C07284=1082.092,-4.857,441.669,174.077,19.888,153.353
C07285=1082.085,-5.106,441.682,174.075,19.886,153.353
C07286=1082.080,-5.356,441.696,174.074,19.884,153.352
C07287=1082.073,-5.606,441.710,174.073,19.882,153.352
C07288=1082.068,-5.855,441.724,174.072,19.880,153.352
C07289=1082.061,-6.105,441.737,174.069,19.877,153.352
C07290=1082.056,-6.354,441.751,174.068,19.875,153.352
C07291=1082.050,-6.603,441.764,174.067,19.873,153.352
C07292=1082.044,-6.853,441.778,174.066,19.871,153.351
C07293=1082.037,-7.103,441.792,174.064,19.870,153.351
C07294=1082.032,-7.352,441.806,174.062,19.867,153.351
C07295=1082.026,-7.602,441.819,174.061,19.865,153.351
C07296=1082.020,-7.851,441.833,174.060,19.863,153.351
C07297=1082.015,-8.102,441.846,174.058,19.861,153.351
C07298=1082.009,-8.351,441.859,174.056,19.859,153.351
C07299=1082.003,-8.600,441.873,174.055,19.857,153.350
C07300=1081.997,-8.850,441.886,174.054,19.855,153.350
C07301=1081.991,-9.100,441.901,174.052,19.853,153.350
C07302=1081.985,-9.349,441.914,174.051,19.851,153.350
C07303=1081.979,-9.599,441.928,174.049,19.848,153.350
C07304=1081.973,-9.848,441.941,174.048,19.846,153.350
C07305=1081.968,-10.098,441.954,174.046,19.845,153.350
C07306=1081.962,-10.347,441.967,174.045,19.843,153.349
C07307=1081.956,-10.597,441.981,174.043,19.840,153.349
C07308=1081.950,-10.846,441.994,174.042,19.838,153.349
C07309=1081.945,-11.096,442.008,174.041,19.836,153.349
C07310=1081.938,-11.345,442.022,174.039,19.834,153.349
C07311=1081.932,-11.595,442.034,174.038,19.832,153.349
C07312=1081.927,-11.845,442.048,174.036,19.830,153.348
C07313=1081.920,-12.095,442.062,174.035,19.828,153.348
C07314=1081.915,-12.344,442.076,174.033,19.826,153.348
C07315=1081.908,-12.593,442.089,174.032,19.824,153.348
C07316=1081.903,-12.844,442.102,174.031,19.822,153.348
C07317=1081.897,-13.093,442.115,174.029,19.820,153.348
C07318=1081.892,-13.342,442.129,174.027,19.818,153.348
C07319=1081.885,-13.592,442.142,174.026,19.816,153.347
C07320=1081.880,-13.842,442.156,174.025,19.814,153.347
C07321=1081.874,-14.091,442.169,174.023,19.811,153.347
C07322=1081.869,-14.341,442.183,174.021,19.809,153.347
C07323=1081.862,-14.590,442.196,174.020,19.807,153.347
C07324=1081.856,-14.840,442.208,174.019,19.805,153.347
C07325=1081.851,-15.089,442.222,174.018,19.803,153.346
C07326=1081.845,-15.339,442.236,174.016,19.801,153.346
C07327=1081.839,-15.589,442.248,174.014,19.799,153.346
C07328=1081.833,-15.838,442.262,174.013,19.797,153.346
C07329=1081.827,-16.087,442.275,174.012,19.795,153.346
C07330=1081.821,-16.337,442.288,174.010,19.793,153.346
C07331=1081.816,-16.587,442.302,174.008,19.791,153.346
C07332=1081.809,-16.860,442.316,174.007,19.789,153.345
C07333=1081.802,-17.135,442.331,174.006,19.787,153.345
C07334=1081.796,-17.409,442.345,174.004,19.784,153.345
C07335=1081.789,-17.683,442.360,174.002,19.782,153.345
C07336=1081.783,-17.933,442.372,174.001,19.780,153.345
C07337=1081.777,-18.182,442.386,173.999,19.778,153.345
C07338=1081.772,-18.431,442.399,173.998,19.776,153.345
C07339=1081.766,-18.681,442.412,173.996,19.774,153.344
C07340=1081.760,-18.931,442.425,173.995,19.772,153.344
C07341=1081.754,-19.180,442.438,173.994,19.770,153.344
C07342=1081.748,-19.430,442.452,173.992,19.768,153.344
C07343=1081.742,-19.680,442.464,173.990,19.766,153.344
C07344=1081.736,-19.929,442.477,173.989,19.764,153.344
C07345=1081.730,-20.178,442.491,173.988,19.762,153.344
C07346=1081.724,-20.428,442.503,173.987,19.760,153.343
C07347=1081.719,-20.678,442.517,173.984,19.758,153.343
C07348=1081.713,-20.928,442.530,173.983,19.756,153.343
C07349=1081.706,-21.177,442.543,173.982,19.754,153.343
C07350=1081.701,-21.427,442.556,173.980,19.752,153.343
C07351=1081.695,-21.677,442.569,173.979,19.750,153.343
C07352=1081.689,-21.926,442.582,173.978,19.748,153.343
C07353=1081.683,-22.176,442.595,173.976,19.746,153.342
C07354=1081.677,-22.426,442.608,173.974,19.744,153.342
C07355=1081.671,-22.675,442.621,173.973,19.742,153.342
C07356=1081.666,-22.925,442.634,173.972,19.740,153.342
C07357=1081.659,-23.174,442.647,173.971,19.738,153.342
C07358=1081.654,-23.424,442.660,173.969,19.736,153.342
C07359=1081.647,-23.673,442.673,173.967,19.734,153.342
C07360=1081.642,-23.923,442.685,173.966,19.732,153.342
C07361=1081.636,-24.172,442.699,173.965,19.730,153.341
C07362=1081.631,-24.422,442.712,173.963,19.728,153.341
C07363=1081.625,-24.672,442.724,173.961,19.725,153.341
C07364=1081.618,-24.921,442.738,173.960,19.723,153.341
C07365=1081.613,-25.171,442.750,173.958,19.722,153.341
C07366=1081.606,-25.420,442.764,173.957,19.720,153.341
C07367=1081.600,-25.670,442.776,173.956,19.718,153.341
C07368=1081.595,-25.920,442.789,173.955,19.716,153.340
C07369=1081.590,-26.169,442.802,173.953,19.713,153.340
C07370=1081.584,-26.419,442.815,173.951,19.712,153.340
C07371=1081.578,-26.668,442.828,173.950,19.710,153.340
C07372=1081.572,-26.918,442.841,173.949,19.708,153.340
C07373=1081.566,-27.168,442.853,173.947,19.706,153.340
C07374=1081.560,-27.417,442.866,173.946,19.704,153.340
C07375=1081.554,-27.667,442.879,173.944,19.702,153.340
C07376=1081.548,-27.917,442.891,173.943,19.700,153.339
C07377=1081.541,-28.166,442.905,173.941,19.698,153.339
C07378=1081.536,-28.415,442.917,173.940,19.696,153.339
C07379=1081.530,-28.665,442.929,173.939,19.694,153.339
C07380=1081.524,-28.915,442.943,173.937,19.692,153.339
C07381=1081.518,-29.164,442.955,173.935,19.690,153.339
C07382=1081.512,-29.414,442.968,173.934,19.688,153.339
C07383=1081.506,-29.664,442.980,173.933,19.686,153.338
C07384=1081.500,-29.913,442.994,173.931,19.684,153.338
C07385=1081.494,-30.163,443.006,173.930,19.683,153.338
C07386=1081.488,-30.413,443.019,173.929,19.681,153.338
C07387=1081.483,-30.662,443.032,173.927,19.678,153.338
C07388=1081.477,-30.912,443.044,173.925,19.677,153.338
C07389=1081.471,-31.162,443.057,173.924,19.675,153.338
C07390=1081.465,-31.411,443.069,173.923,19.673,153.338
C07391=1081.459,-31.661,443.082,173.921,19.671,153.338
C07392=1081.452,-31.910,443.095,173.920,19.669,153.337
C07393=1081.447,-32.159,443.107,173.918,19.667,153.337
C07394=1081.441,-32.409,443.119,173.916,19.665,153.337
C07395=1081.435,-32.659,443.132,173.915,19.663,153.337
C07396=1081.428,-32.933,443.146,173.914,19.661,153.337
C07397=1081.422,-33.206,443.160,173.912,19.659,153.337
C07398=1081.416,-33.479,443.173,173.910,19.657,153.337
C07399=1081.409,-33.752,443.188,173.909,19.655,153.336
C07400=1081.403,-34.002,443.200,173.908,19.653,153.336
C07401=1081.398,-34.251,443.212,173.906,19.651,153.336
C07402=1081.392,-34.501,443.225,173.904,19.649,153.336
C07403=1081.386,-34.751,443.237,173.903,19.647,153.336
C07404=1081.379,-35.001,443.249,173.902,19.645,153.336
C07405=1081.373,-35.250,443.263,173.900,19.643,153.336
C07406=1081.368,-35.499,443.275,173.899,19.642,153.336
C07407=1081.362,-35.749,443.287,173.897,19.639,153.336
C07408=1081.356,-35.999,443.300,173.896,19.637,153.335
C07409=1081.350,-36.249,443.312,173.894,19.636,153.335
C07410=1081.345,-36.498,443.325,173.893,19.634,153.335
C07411=1081.339,-36.748,443.337,173.892,19.632,153.335
C07412=1081.333,-36.998,443.350,173.890,19.630,153.335
C07413=1081.326,-37.247,443.362,173.889,19.628,153.335
C07414=1081.321,-37.496,443.374,173.887,19.626,153.335
C07415=1081.315,-37.746,443.386,173.885,19.624,153.335
C07416=1081.309,-37.996,443.399,173.884,19.622,153.334
C07417=1081.303,-38.245,443.412,173.883,19.620,153.334
C07418=1081.298,-38.495,443.424,173.881,19.618,153.334
C07419=1081.291,-38.744,443.436,173.880,19.616,153.334
C07420=1081.285,-38.994,443.449,173.879,19.614,153.334
C07421=1081.279,-39.244,443.462,173.877,19.612,153.334
C07422=1081.274,-39.493,443.474,173.875,19.610,153.334
C07423=1081.267,-39.743,443.486,173.874,19.609,153.334
C07424=1081.261,-39.993,443.498,173.873,19.607,153.334
C07425=1081.255,-40.243,443.511,173.871,19.605,153.334
C07426=1081.249,-40.491,443.522,173.870,19.603,153.333
C07427=1081.243,-40.741,443.535,173.869,19.601,153.333
C07428=1081.238,-40.992,443.547,173.867,19.600,153.333
C07429=1081.231,-41.241,443.559,173.865,19.597,153.333
C07430=1081.226,-41.491,443.571,173.864,19.596,153.333
C07431=1081.220,-41.740,443.583,173.862,19.594,153.333
C07432=1081.213,-41.990,443.595,173.861,19.592,153.333
C07433=1081.207,-42.240,443.608,173.860,19.590,153.333
C07434=1081.202,-42.489,443.620,173.858,19.589,153.333
C07435=1081.195,-42.739,443.632,173.857,19.587,153.332
C07436=1081.190,-42.989,443.645,173.855,19.584,153.332
C07437=1081.184,-43.238,443.657,173.853,19.583,153.332
C07438=1081.178,-43.487,443.669,173.852,19.581,153.332
C07439=1081.172,-43.737,443.681,173.851,19.579,153.332
C07440=1081.167,-43.987,443.693,173.849,19.577,153.332
C07441=1081.160,-44.237,443.705,173.848,19.576,153.332
C07442=1081.154,-44.486,443.717,173.847,19.574,153.332
C07443=1081.148,-44.736,443.730,173.845,19.572,153.332
C07444=1081.142,-44.985,443.742,173.844,19.570,153.331
C07445=1081.136,-45.235,443.754,173.842,19.568,153.331
C07446=1081.130,-45.485,443.766,173.840,19.566,153.331
C07447=1081.125,-45.734,443.778,173.839,19.565,153.331
C07448=1081.119,-45.984,443.790,173.838,19.563,153.331
C07449=1081.112,-46.234,443.802,173.836,19.561,153.331
C07450=1081.107,-46.483,443.814,173.835,19.559,153.331
C07451=1081.100,-46.733,443.826,173.834,19.558,153.331
C07452=1081.095,-46.982,443.838,173.832,19.556,153.331
C07453=1081.089,-47.232,443.850,173.830,19.553,153.331
C07454=1081.083,-47.482,443.862,173.829,19.552,153.331
C07455=1081.077,-47.731,443.874,173.828,19.550,153.330
C07456=1081.072,-47.982,443.886,173.826,19.548,153.330
C07457=1081.065,-48.231,443.898,173.825,19.546,153.330
C07458=1081.060,-48.480,443.910,173.823,19.545,153.330
C07459=1081.053,-48.730,443.922,173.822,19.543,153.330
C07460=1081.047,-49.004,443.935,173.820,19.541,153.330
C07461=1081.040,-49.278,443.948,173.819,19.539,153.330
C07462=1081.034,-49.551,443.962,173.817,19.537,153.330
C07463=1081.027,-49.825,443.975,173.816,19.535,153.330
C07464=1081.022,-50.074,443.987,173.814,19.533,153.329
C07465=1081.016,-50.324,443.999,173.812,19.531,153.329
C07466=1081.011,-50.574,444.010,173.811,19.530,153.329
C07467=1081.004,-50.823,444.022,173.810,19.527,153.329
C07468=1080.997,-51.073,444.034,173.808,19.526,153.329
C07469=1080.992,-51.322,444.046,173.807,19.524,153.329
C07470=1080.986,-51.572,444.058,173.805,19.522,153.329
C07471=1080.979,-51.822,444.069,173.804,19.521,153.329
C07472=1080.974,-52.072,444.081,173.803,19.519,153.329
C07473=1080.967,-52.321,444.093,173.801,19.517,153.329
C07474=1080.961,-52.571,444.105,173.799,19.515,153.329
C07475=1080.955,-52.820,444.116,173.798,19.513,153.329
C07476=1080.949,-53.070,444.128,173.796,19.512,153.329
C07477=1080.942,-53.320,444.140,173.795,19.510,153.329
C07478=1080.937,-53.569,444.151,173.794,19.508,153.328
C07479=1080.931,-53.819,444.164,173.792,19.507,153.328
C07480=1080.925,-54.069,444.175,173.791,19.505,153.328
C07481=1080.918,-54.318,444.187,173.789,19.503,153.328
C07482=1080.912,-54.568,444.199,173.788,19.502,153.328
C07483=1080.907,-54.817,444.210,173.786,19.500,153.328
C07484=1080.900,-55.067,444.222,173.785,19.499,153.328
C07485=1080.894,-55.317,444.233,173.784,19.497,153.328
C07486=1080.888,-55.566,444.245,173.781,19.495,153.328
C07487=1080.882,-55.817,444.257,173.780,19.493,153.328
C07488=1080.876,-56.065,444.268,173.779,19.491,153.328
C07489=1080.870,-56.315,444.281,173.777,19.490,153.328
C07490=1080.864,-56.565,444.292,173.776,19.488,153.328
C07491=1080.858,-56.814,444.304,173.774,19.486,153.327
C07492=1080.851,-57.065,444.315,173.773,19.485,153.327
C07493=1080.846,-57.314,444.327,173.772,19.483,153.327
C07494=1080.840,-57.564,444.338,173.770,19.482,153.327
C07495=1080.834,-57.813,444.350,173.769,19.480,153.327
C07496=1080.827,-58.063,444.361,173.767,19.478,153.327
C07497=1080.822,-58.312,444.373,173.766,19.477,153.327
C07498=1080.816,-58.562,444.385,173.765,19.475,153.327
C07499=1080.810,-58.812,444.395,173.762,19.473,153.327
C07500=1080.803,-59.061,444.407,173.761,19.471,153.327
C07501=1080.798,-59.312,444.419,173.759,19.470,153.327
C07502=1080.792,-59.561,444.431,173.758,19.468,153.327
C07503=1080.785,-59.811,444.442,173.757,19.466,153.327
C07504=1080.779,-60.060,444.454,173.755,19.465,153.327
C07505=1080.774,-60.310,444.465,173.754,19.463,153.327
C07506=1080.768,-60.559,444.477,173.753,19.461,153.327
C07507=1080.761,-60.809,444.488,173.751,19.460,153.326
C07508=1080.756,-61.059,444.499,173.750,19.458,153.326
C07509=1080.750,-61.309,444.512,173.748,19.457,153.326
C07510=1080.744,-61.558,444.523,173.747,19.455,153.326
C07511=1080.737,-61.808,444.535,173.745,19.453,153.326
C07512=1080.731,-62.057,444.545,173.744,19.452,153.326
C07513=1080.725,-62.308,444.557,173.742,19.450,153.326
C07514=1080.720,-62.557,444.569,173.740,19.448,153.326
C07515=1080.713,-62.807,444.580,173.739,19.446,153.326
C07516=1080.708,-63.056,444.591,173.737,19.445,153.326
C07517=1080.702,-63.305,444.603,173.736,19.443,153.326
C07518=1080.695,-63.556,444.614,173.735,19.441,153.326
C07519=1080.690,-63.805,444.625,173.733,19.440,153.326
C07520=1080.684,-64.055,444.637,173.732,19.438,153.326
C07521=1080.678,-64.304,444.648,173.730,19.437,153.326
C07522=1080.672,-64.555,444.659,173.729,19.435,153.326
C07523=1080.666,-64.803,444.671,173.728,19.433,153.326
C07524=1080.660,-65.079,444.683,173.726,19.432,153.325
C07525=1080.653,-65.354,444.696,173.724,19.430,153.326
C07526=1080.646,-65.629,444.708,173.723,19.428,153.325
C07527=1080.640,-65.904,444.721,173.721,19.426,153.325
C07528=1080.634,-66.153,444.732,173.720,19.425,153.325
C07529=1080.627,-66.403,444.744,173.718,19.423,153.325
C07530=1080.622,-66.652,444.754,173.717,19.421,153.325
C07531=1080.615,-66.903,444.766,173.716,19.420,153.325
C07532=1080.610,-67.152,444.777,173.714,19.418,153.325
C07533=1080.604,-67.401,444.789,173.713,19.417,153.325
C07534=1080.598,-67.652,444.800,173.711,19.415,153.325
C07535=1080.592,-67.901,444.811,173.710,19.414,153.325
C07536=1080.586,-68.151,444.822,173.708,19.412,153.325
C07537=1080.580,-68.401,444.833,173.707,19.410,153.325
C07538=1080.574,-68.650,444.845,173.705,19.408,153.325
C07539=1080.568,-68.900,444.856,173.703,19.407,153.325
C07540=1080.563,-69.150,444.867,173.702,19.405,153.325
C07541=1080.557,-69.399,444.878,173.700,19.404,153.325
C07542=1080.551,-69.649,444.889,173.699,19.401,153.324
C07543=1080.545,-69.899,444.900,173.698,19.400,153.324
C07544=1080.539,-70.148,444.912,173.696,19.398,153.324
C07545=1080.533,-70.398,444.923,173.695,19.397,153.324
C07546=1080.527,-70.647,444.934,173.693,19.395,153.324
C07547=1080.521,-70.897,444.945,173.692,19.394,153.324
C07548=1080.515,-71.147,444.957,173.690,19.392,153.324
C07549=1080.510,-71.397,444.968,173.689,19.390,153.324
C07550=1080.504,-71.646,444.978,173.687,19.389,153.324
C07551=1080.498,-71.896,444.990,173.686,19.387,153.324
C07552=1080.492,-72.145,445.001,173.685,19.386,153.324
C07553=1080.486,-72.395,445.012,173.683,19.384,153.324
C07554=1080.479,-72.645,445.023,173.682,19.383,153.324
C07555=1080.474,-72.894,445.034,173.680,19.381,153.324
C07556=1080.468,-73.144,445.045,173.679,19.380,153.324
C07557=1080.462,-73.393,445.056,173.677,19.378,153.324
C07558=1080.456,-73.644,445.067,173.676,19.376,153.324
C07559=1080.451,-73.893,445.079,173.675,19.375,153.324
C07560=1080.445,-74.143,445.090,173.673,19.373,153.324
C07561=1080.438,-74.393,445.100,173.672,19.372,153.324
C07562=1080.432,-74.642,445.111,173.670,19.370,153.324
C07563=1080.427,-74.892,445.122,173.669,19.369,153.324
C07564=1080.420,-75.142,445.133,173.667,19.367,153.324
C07565=1080.415,-75.392,445.144,173.666,19.366,153.324
C07566=1080.409,-75.641,445.155,173.664,19.364,153.324
C07567=1080.402,-75.891,445.166,173.663,19.363,153.323
C07568=1080.397,-76.141,445.177,173.661,19.361,153.323
C07569=1080.390,-76.390,445.187,173.660,19.360,153.323
C07570=1080.384,-76.640,445.199,173.658,19.359,153.324
C07571=1080.378,-76.890,445.210,173.657,19.357,153.324
C07572=1080.372,-77.139,445.220,173.655,19.356,153.323
C07573=1080.366,-77.389,445.232,173.654,19.354,153.323
C07574=1080.360,-77.639,445.243,173.652,19.353,153.323
C07575=1080.355,-77.888,445.253,173.651,19.351,153.323
C07576=1080.349,-78.138,445.264,173.649,19.350,153.323
C07577=1080.342,-78.388,445.275,173.648,19.348,153.323
C07578=1080.336,-78.637,445.286,173.646,19.347,153.323
C07579=1080.330,-78.887,445.297,173.645,19.345,153.323
C07580=1080.324,-79.137,445.307,173.643,19.344,153.323
C07581=1080.319,-79.387,445.318,173.642,19.342,153.323
C07582=1080.313,-79.636,445.329,173.641,19.341,153.323
C07583=1080.306,-79.886,445.339,173.639,19.339,153.323
C07584=1080.300,-80.136,445.351,173.638,19.338,153.323
C07585=1080.294,-80.385,445.361,173.636,19.337,153.323
C07586=1080.289,-80.635,445.372,173.634,19.335,153.323
C07587=1080.281,-80.885,445.383,173.633,19.334,153.323
C07588=1080.276,-81.162,445.394,173.631,19.332,153.323
C07589=1080.268,-81.439,445.406,173.629,19.330,153.323
C07590=1080.261,-81.716,445.419,173.628,19.329,153.323
C07591=1080.255,-81.993,445.430,173.626,19.327,153.323
C07592=1080.248,-82.243,445.441,173.625,19.326,153.323
C07593=1080.243,-82.493,445.452,173.623,19.325,153.323
C07594=1080.236,-82.742,445.462,173.622,19.323,153.323
C07595=1080.230,-82.991,445.473,173.620,19.322,153.323
C07596=1080.224,-83.242,445.483,173.618,19.321,153.323
C07597=1080.218,-83.491,445.494,173.617,19.319,153.323
C07598=1080.212,-83.741,445.505,173.615,19.318,153.323
C07599=1080.206,-83.991,445.516,173.614,19.316,153.323
C07600=1080.199,-84.240,445.526,173.613,19.315,153.323
C07601=1080.194,-84.490,445.536,173.611,19.314,153.323
C07602=1080.188,-84.740,445.547,173.609,19.312,153.323
C07603=1080.181,-84.990,445.558,173.608,19.311,153.323
C07604=1080.175,-85.239,445.569,173.606,19.309,153.323
C07605=1080.169,-85.489,445.578,173.605,19.308,153.323
C07606=1080.164,-85.738,445.589,173.603,19.307,153.323
C07607=1080.157,-85.989,445.600,173.603,19.306,153.323
C07608=1080.151,-86.238,445.611,173.601,19.304,153.323
C07609=1080.145,-86.488,445.621,173.600,19.303,153.323
C07610=1080.139,-86.737,445.631,173.598,19.302,153.323
C07611=1080.133,-86.987,445.642,173.597,19.300,153.323
C07612=1080.127,-87.237,445.652,173.595,19.299,153.323
C07613=1080.121,-87.487,445.663,173.593,19.298,153.323
C07614=1080.115,-87.736,445.674,173.592,19.296,153.323
C07615=1080.109,-87.986,445.683,173.590,19.295,153.323
C07616=1080.103,-88.235,445.694,173.589,19.294,153.323
C07617=1080.097,-88.486,445.705,173.587,19.292,153.323
C07618=1080.090,-88.735,445.715,173.586,19.291,153.323
C07619=1080.085,-88.985,445.726,173.584,19.290,153.323
C07620=1080.078,-89.234,445.736,173.583,19.288,153.323
C07621=1080.073,-89.484,445.746,173.581,19.287,153.323
C07622=1080.066,-89.733,445.756,173.579,19.286,153.324
C07623=1080.060,-89.984,445.768,173.578,19.284,153.324
C07624=1080.054,-90.234,445.778,173.577,19.283,153.323
C07625=1080.048,-90.483,445.788,173.575,19.282,153.324
C07626=1080.043,-90.733,445.798,173.573,19.280,153.324
C07627=1080.036,-90.982,445.809,173.572,19.279,153.324
C07628=1080.030,-91.232,445.819,173.571,19.278,153.324
C07629=1080.024,-91.482,445.829,173.570,19.277,153.324
C07630=1080.018,-91.732,445.840,173.568,19.275,153.324
C07631=1080.012,-91.981,445.850,173.566,19.275,153.324
C07632=1080.006,-92.231,445.861,173.565,19.273,153.324
C07633=1080.000,-92.480,445.872,173.564,19.272,153.324
C07634=1079.994,-92.730,445.881,173.562,19.271,153.324
C07635=1079.988,-92.980,445.892,173.560,19.269,153.324
C07636=1079.982,-93.229,445.902,173.559,19.268,153.324
C07637=1079.976,-93.480,445.913,173.557,19.267,153.324
C07638=1079.970,-93.729,445.922,173.556,19.265,153.324
C07639=1079.964,-93.979,445.933,173.554,19.264,153.324
C07640=1079.958,-94.229,445.943,173.553,19.263,153.324
C07641=1079.952,-94.478,445.954,173.551,19.261,153.324
C07642=1079.946,-94.728,445.963,173.549,19.260,153.324
C07643=1079.940,-94.977,445.974,173.548,19.259,153.324
C07644=1079.934,-95.227,445.984,173.547,19.258,153.324
C07645=1079.928,-95.477,445.995,173.546,19.257,153.324
C07646=1079.922,-95.727,446.004,173.544,19.255,153.324
C07647=1079.916,-95.976,446.015,173.542,19.254,153.324
C07648=1079.910,-96.226,446.025,173.541,19.253,153.324
C07649=1079.905,-96.476,446.035,173.539,19.252,153.324
C07650=1079.898,-96.726,446.045,173.538,19.250,153.324
C07651=1079.892,-96.976,446.056,173.536,19.249,153.324
C07652=1079.885,-97.255,446.067,173.535,19.248,153.324
C07653=1079.879,-97.535,446.078,173.533,19.246,153.324
C07654=1079.872,-97.815,446.090,173.531,19.245,153.324
C07655=1079.865,-98.094,446.101,173.530,19.244,153.324
C07656=1079.859,-98.345,446.111,173.528,19.243,153.324
C07657=1079.853,-98.594,446.121,173.527,19.241,153.324
C07658=1079.847,-98.844,446.131,173.525,19.240,153.324
C07659=1079.840,-99.093,446.141,173.523,19.239,153.325
C07660=1079.835,-99.343,446.151,173.522,19.238,153.325
C07661=1079.828,-99.592,446.162,173.520,19.237,153.325
C07662=1079.822,-99.842,446.171,173.519,19.235,153.325
C07663=1079.816,-100.091,446.182,173.517,19.234,153.325
C07664=1079.810,-100.341,446.192,173.516,19.233,153.325
C07665=1079.804,-100.590,446.202,173.515,19.232,153.325
C07666=1079.798,-100.840,446.212,173.513,19.231,153.325
C07667=1079.791,-101.090,446.221,173.512,19.230,153.325
C07668=1079.786,-101.339,446.232,173.510,19.229,153.325
C07669=1079.780,-101.589,446.242,173.508,19.227,153.325
C07670=1079.773,-101.839,446.251,173.507,19.226,153.325
C07671=1079.768,-102.088,446.262,173.505,19.225,153.325
C07672=1079.761,-102.338,446.272,173.504,19.224,153.325
C07673=1079.755,-102.588,446.281,173.502,19.223,153.325
C07674=1079.749,-102.837,446.291,173.500,19.221,153.325
C07675=1079.743,-103.087,446.302,173.500,19.221,153.325
C07676=1079.737,-103.337,446.311,173.498,19.220,153.325
C07677=1079.731,-103.587,446.321,173.496,19.218,153.325
C07678=1079.725,-103.836,446.331,173.495,19.217,153.326
C07679=1079.719,-104.086,446.341,173.493,19.216,153.326
C07680=1079.713,-104.336,446.351,173.491,19.215,153.326
C07681=1079.707,-104.586,446.360,173.490,19.214,153.326
C07682=1079.700,-104.835,446.371,173.488,19.213,153.326
C07683=1079.695,-105.085,446.381,173.487,19.212,153.326
C07684=1079.689,-105.335,446.390,173.486,19.211,153.326
C07685=1079.683,-105.585,446.400,173.484,19.210,153.326
C07686=1079.676,-105.834,446.409,173.483,19.209,153.326
C07687=1079.671,-106.084,446.420,173.481,19.208,153.326
C07688=1079.664,-106.334,446.430,173.479,19.207,153.326
C07689=1079.658,-106.584,446.439,173.477,19.206,153.326
C07690=1079.652,-106.833,446.449,173.476,19.204,153.326
C07691=1079.646,-107.083,446.459,173.475,19.204,153.326
C07692=1079.640,-107.333,446.469,173.473,19.203,153.327
C07693=1079.634,-107.582,446.479,173.472,19.201,153.326
C07694=1079.628,-107.832,446.489,173.470,19.200,153.327
C07695=1079.622,-108.082,446.498,173.469,19.199,153.327
C07696=1079.616,-108.332,446.508,173.467,19.198,153.327
C07697=1079.609,-108.582,446.517,173.465,19.197,153.327
C07698=1079.603,-108.831,446.528,173.464,19.196,153.327
C07699=1079.597,-109.081,446.537,173.463,19.195,153.327
C07700=1079.591,-109.330,446.547,173.461,19.194,153.327
C07701=1079.585,-109.581,446.557,173.459,19.193,153.327
C07702=1079.579,-109.830,446.566,173.458,19.192,153.327
C07703=1079.573,-110.080,446.576,173.456,19.191,153.327
C07704=1079.567,-110.330,446.586,173.455,19.190,153.327
C07705=1079.560,-110.580,446.595,173.453,19.189,153.328
C07706=1079.554,-110.829,446.605,173.452,19.188,153.328
C07707=1079.548,-111.079,446.615,173.450,19.187,153.328
C07708=1079.542,-111.328,446.625,173.449,19.186,153.328
C07709=1079.535,-111.578,446.634,173.447,19.185,153.328
C07710=1079.529,-111.828,446.644,173.445,19.184,153.328
C07711=1079.524,-112.077,446.653,173.444,19.183,153.328
C07712=1079.518,-112.327,446.662,173.443,19.183,153.328
C07713=1079.511,-112.577,446.672,173.441,19.182,153.328
C07714=1079.505,-112.827,446.682,173.439,19.181,153.328
C07715=1079.500,-113.077,446.692,173.438,19.180,153.328
C07716=1079.492,-113.353,446.702,173.436,19.179,153.329
C07717=1079.486,-113.629,446.712,173.435,19.177,153.329
C07718=1079.479,-113.905,446.723,173.433,19.176,153.329
C07719=1079.472,-114.182,446.734,173.431,19.175,153.329
C07720=1079.466,-114.432,446.744,173.429,19.174,153.329
C07721=1079.460,-114.682,446.753,173.428,19.173,153.329
C07722=1079.454,-114.932,446.763,173.426,19.172,153.329
C07723=1079.448,-115.181,446.772,173.425,19.172,153.329
C07724=1079.442,-115.431,446.782,173.424,19.171,153.329
C07725=1079.436,-115.680,446.791,173.422,19.170,153.329
C07726=1079.430,-115.930,446.801,173.420,19.169,153.330
C07727=1079.423,-116.180,446.810,173.418,19.168,153.330
C07728=1079.417,-116.430,446.820,173.417,19.167,153.330
C07729=1079.411,-116.680,446.829,173.416,19.166,153.330
C07730=1079.405,-116.930,446.838,173.414,19.165,153.330
C07731=1079.398,-117.180,446.847,173.412,19.164,153.330
C07732=1079.392,-117.429,446.857,173.411,19.164,153.330
C07733=1079.387,-117.678,446.866,173.409,19.163,153.330
C07734=1079.380,-117.928,446.876,173.407,19.162,153.330
C07735=1079.374,-118.178,446.885,173.406,19.161,153.331
C07736=1079.368,-118.428,446.895,173.405,19.160,153.331
C07737=1079.362,-118.678,446.904,173.403,19.159,153.331
C07738=1079.356,-118.927,446.914,173.401,19.158,153.331
C07739=1079.350,-119.177,446.923,173.400,19.157,153.331
C07740=1079.344,-119.428,446.932,173.399,19.157,153.331
C07741=1079.337,-119.676,446.941,173.397,19.156,153.331
C07742=1079.331,-119.926,446.950,173.395,19.155,153.331
C07743=1079.325,-120.176,446.960,173.394,19.154,153.331
C07744=1079.319,-120.426,446.970,173.392,19.153,153.332
C07745=1079.313,-120.676,446.979,173.391,19.152,153.332
C07746=1079.307,-120.925,446.989,173.389,19.151,153.332
C07747=1079.301,-121.175,446.997,173.388,19.150,153.332
C07748=1079.295,-121.425,447.007,173.386,19.150,153.332
C07749=1079.288,-121.674,447.016,173.384,19.149,153.332
C07750=1079.282,-121.924,447.025,173.383,19.148,153.332
C07751=1079.276,-122.174,447.035,173.381,19.148,153.332
C07752=1079.270,-122.424,447.044,173.380,19.147,153.333
C07753=1079.264,-122.674,447.053,173.378,19.146,153.333
C07754=1079.258,-122.923,447.063,173.376,19.145,153.333
C07755=1079.251,-123.173,447.072,173.376,19.144,153.333
C07756=1079.245,-123.423,447.081,173.374,19.144,153.333
C07757=1079.239,-123.673,447.090,173.372,19.143,153.333
C07758=1079.233,-123.923,447.099,173.370,19.142,153.333
C07759=1079.228,-124.172,447.109,173.368,19.141,153.333
C07760=1079.221,-124.422,447.118,173.368,19.140,153.334
C07761=1079.215,-124.672,447.127,173.366,19.139,153.334
C07762=1079.209,-124.922,447.136,173.364,19.139,153.334
C07763=1079.202,-125.171,447.146,173.362,19.138,153.334
C07764=1079.196,-125.420,447.154,173.361,19.137,153.334
C07765=1079.190,-125.671,447.163,173.360,19.136,153.334
C07766=1079.184,-125.920,447.173,173.358,19.135,153.334
C07767=1079.178,-126.170,447.182,173.356,19.135,153.335
C07768=1079.171,-126.420,447.191,173.354,19.134,153.335
C07769=1079.166,-126.669,447.200,173.353,19.134,153.335
C07770=1079.160,-126.919,447.209,173.352,19.133,153.335
C07771=1079.153,-127.169,447.218,173.350,19.132,153.335
C07772=1079.147,-127.419,447.227,173.348,19.131,153.335
C07773=1079.141,-127.670,447.236,173.346,19.130,153.335
C07774=1079.135,-127.919,447.246,173.346,19.130,153.335
C07775=1079.130,-128.169,447.255,173.344,19.129,153.336
C07776=1079.128,-128.424,447.266,173.343,19.127,153.335
C07777=1079.129,-128.679,447.278,173.342,19.124,153.335
C07778=1079.134,-128.932,447.291,173.342,19.119,153.334
C07779=1079.141,-129.184,447.305,173.342,19.115,153.333
C07780=1078.744,-129.205,447.160,173.297,19.238,153.364
C07781=1078.736,-128.954,447.147,173.297,19.243,153.365
C07782=1078.732,-128.701,447.133,173.298,19.247,153.366
C07783=1078.730,-128.446,447.121,173.299,19.250,153.366
C07784=1078.732,-128.191,447.109,173.299,19.252,153.366
C07785=1078.736,-127.941,447.100,173.301,19.253,153.366
C07786=1078.743,-127.691,447.091,173.302,19.254,153.366
C07787=1078.748,-127.441,447.082,173.304,19.255,153.366
C07788=1078.755,-127.191,447.073,173.306,19.256,153.366
C07789=1078.761,-126.941,447.064,173.307,19.256,153.366
C07790=1078.767,-126.692,447.055,173.308,19.257,153.366
C07791=1078.773,-126.442,447.045,173.310,19.258,153.365
C07792=1078.779,-126.192,447.037,173.312,19.259,153.365
C07793=1078.786,-125.942,447.027,173.314,19.259,153.365
C07794=1078.792,-125.692,447.018,173.315,19.260,153.365
C07795=1078.798,-125.443,447.010,173.316,19.261,153.365
C07796=1078.804,-125.193,447.000,173.318,19.262,153.365
C07797=1078.810,-124.943,446.991,173.320,19.262,153.364
C07798=1078.816,-124.694,446.981,173.321,19.263,153.364
C07799=1078.823,-124.444,446.973,173.323,19.264,153.364
C07800=1078.829,-124.194,446.963,173.324,19.265,153.364
C07801=1078.835,-123.945,446.954,173.326,19.266,153.364
C07802=1078.841,-123.695,446.945,173.328,19.267,153.364
C07803=1078.847,-123.444,446.936,173.329,19.267,153.364
C07804=1078.853,-123.195,446.926,173.330,19.268,153.364
C07805=1078.860,-122.945,446.917,173.332,19.268,153.363
C07806=1078.865,-122.696,446.908,173.334,19.269,153.363
C07807=1078.872,-122.446,446.899,173.336,19.270,153.363
C07808=1078.877,-122.196,446.890,173.337,19.271,153.363
C07809=1078.884,-121.946,446.880,173.338,19.272,153.363
C07810=1078.890,-121.696,446.871,173.340,19.273,153.363
C07811=1078.897,-121.447,446.862,173.342,19.274,153.363
C07812=1078.902,-121.198,446.852,173.343,19.275,153.363
C07813=1078.908,-120.947,446.844,173.344,19.275,153.363
C07814=1078.914,-120.697,446.834,173.346,19.276,153.363
C07815=1078.920,-120.448,446.824,173.348,19.277,153.362
C07816=1078.927,-120.198,446.815,173.349,19.278,153.362
C07817=1078.933,-119.948,446.805,173.351,19.278,153.362
C07818=1078.939,-119.699,446.797,173.353,19.279,153.362
C07819=1078.945,-119.449,446.787,173.354,19.280,153.362
C07820=1078.951,-119.199,446.778,173.356,19.281,153.362
C07821=1078.957,-118.949,446.769,173.357,19.282,153.362
C07822=1078.963,-118.699,446.759,173.359,19.283,153.362
C07823=1078.970,-118.450,446.750,173.361,19.284,153.361
C07824=1078.976,-118.200,446.740,173.362,19.284,153.361
C07825=1078.982,-117.950,446.730,173.363,19.285,153.361
C07826=1078.988,-117.701,446.721,173.365,19.286,153.361
C07827=1078.994,-117.451,446.712,173.367,19.287,153.361
C07828=1079.000,-117.201,446.702,173.368,19.288,153.361
C07829=1079.007,-116.952,446.693,173.370,19.289,153.361
C07830=1079.013,-116.702,446.684,173.371,19.290,153.361
C07831=1079.019,-116.452,446.675,173.373,19.291,153.361
C07832=1079.025,-116.202,446.665,173.374,19.292,153.361
C07833=1079.031,-115.952,446.656,173.376,19.293,153.360
C07834=1079.037,-115.702,446.646,173.378,19.294,153.360
C07835=1079.044,-115.452,446.636,173.379,19.295,153.360
C07836=1079.049,-115.203,446.627,173.380,19.295,153.360
C07837=1079.055,-114.954,446.618,173.382,19.296,153.360
C07838=1079.061,-114.704,446.608,173.384,19.297,153.360
C07839=1079.068,-114.454,446.599,173.385,19.298,153.360
C07840=1079.074,-114.204,446.589,173.387,19.299,153.360
C07841=1079.080,-113.927,446.578,173.389,19.300,153.360
C07842=1079.088,-113.651,446.568,173.390,19.301,153.359
C07843=1079.094,-113.375,446.557,173.392,19.303,153.359
C07844=1079.101,-113.098,446.546,173.394,19.304,153.359
C07845=1079.107,-112.848,446.536,173.395,19.305,153.359
C07846=1079.113,-112.599,446.527,173.397,19.306,153.359
C07847=1079.119,-112.349,446.517,173.398,19.306,153.359
C07848=1079.125,-112.099,446.508,173.400,19.307,153.359
C07849=1079.131,-111.849,446.498,173.401,19.308,153.359
C07850=1079.138,-111.599,446.489,173.403,19.310,153.359
C07851=1079.144,-111.350,446.479,173.404,19.311,153.359
C07852=1079.150,-111.100,446.469,173.406,19.311,153.359
C07853=1079.156,-110.850,446.460,173.408,19.312,153.358
C07854=1079.162,-110.600,446.450,173.409,19.313,153.358
C07855=1079.168,-110.350,446.441,173.410,19.314,153.358
C07856=1079.174,-110.101,446.432,173.412,19.315,153.358
C07857=1079.180,-109.852,446.421,173.414,19.316,153.358
C07858=1079.186,-109.602,446.411,173.415,19.317,153.358
C07859=1079.192,-109.352,446.402,173.417,19.318,153.358
C07860=1079.198,-109.102,446.392,173.418,19.320,153.358
C07861=1079.204,-108.853,446.382,173.419,19.320,153.358
C07862=1079.211,-108.603,446.373,173.421,19.321,153.358
C07863=1079.217,-108.353,446.363,173.423,19.322,153.358
C07864=1079.223,-108.104,446.353,173.424,19.324,153.358
C07865=1079.229,-107.854,446.343,173.426,19.325,153.358
C07866=1079.236,-107.604,446.334,173.428,19.326,153.358
C07867=1079.241,-107.354,446.324,173.429,19.327,153.357
C07868=1079.247,-107.104,446.314,173.431,19.328,153.357
C07869=1079.253,-106.855,446.305,173.432,19.329,153.357
C07870=1079.260,-106.605,446.294,173.433,19.330,153.357
C07871=1079.266,-106.356,446.285,173.435,19.331,153.357
C07872=1079.271,-106.105,446.275,173.437,19.332,153.357
C07873=1079.278,-105.856,446.265,173.438,19.333,153.357
C07874=1079.284,-105.606,446.255,173.440,19.334,153.357
C07875=1079.290,-105.357,446.245,173.441,19.335,153.357
C07876=1079.296,-105.107,446.236,173.443,19.336,153.357
C07877=1079.302,-104.857,446.225,173.444,19.337,153.357
C07878=1079.308,-104.607,446.216,173.445,19.338,153.357
C07879=1079.315,-104.358,446.206,173.447,19.339,153.357
C07880=1079.321,-104.108,446.196,173.449,19.341,153.357
C07881=1079.326,-103.858,446.186,173.450,19.342,153.357
C07882=1079.332,-103.608,446.176,173.452,19.343,153.356
C07883=1079.339,-103.359,446.166,173.453,19.344,153.356
C07884=1079.345,-103.109,446.156,173.455,19.345,153.356
C07885=1079.350,-102.859,446.146,173.457,19.347,153.356
C07886=1079.357,-102.609,446.137,173.458,19.347,153.356
C07887=1079.363,-102.360,446.126,173.459,19.348,153.356
C07888=1079.369,-102.110,446.116,173.461,19.350,153.356
C07889=1079.375,-101.860,446.107,173.462,19.351,153.356
C07890=1079.382,-101.610,446.096,173.464,19.352,153.356
C07891=1079.388,-101.360,446.086,173.466,19.353,153.356
C07892=1079.393,-101.110,446.076,173.467,19.354,153.356
C07893=1079.400,-100.861,446.066,173.469,19.356,153.356
C07894=1079.406,-100.611,446.056,173.470,19.357,153.356
C07895=1079.411,-100.361,446.046,173.472,19.358,153.356
C07896=1079.418,-100.112,446.036,173.473,19.359,153.356
C07897=1079.424,-99.862,446.026,173.474,19.360,153.356
C07898=1079.430,-99.612,446.016,173.476,19.361,153.356
C07899=1079.436,-99.363,446.006,173.477,19.363,153.356
C07900=1079.442,-99.113,445.996,173.479,19.364,153.356
C07901=1079.449,-98.864,445.986,173.481,19.364,153.355
C07902=1079.454,-98.614,445.976,173.482,19.366,153.356
C07903=1079.460,-98.364,445.966,173.484,19.367,153.355
C07904=1079.467,-98.114,445.956,173.486,19.368,153.355
C07905=1079.474,-97.835,445.944,173.487,19.369,153.355
C07906=1079.480,-97.555,445.934,173.489,19.371,153.355
C07907=1079.487,-97.276,445.922,173.490,19.372,153.355
C07908=1079.494,-96.996,445.911,173.492,19.373,153.355
C07909=1079.499,-96.746,445.901,173.493,19.375,153.355
C07910=1079.506,-96.497,445.890,173.495,19.376,153.355
C07911=1079.511,-96.247,445.880,173.497,19.377,153.355
C07912=1079.518,-95.998,445.870,173.498,19.379,153.355
C07913=1079.524,-95.747,445.859,173.500,19.380,153.355
C07914=1079.530,-95.498,445.849,173.501,19.381,153.355
C07915=1079.536,-95.248,445.839,173.503,19.382,153.355
C07916=1079.541,-94.998,445.828,173.504,19.384,153.355
C07917=1079.548,-94.749,445.818,173.506,19.385,153.355
C07918=1079.553,-94.499,445.808,173.508,19.386,153.355
C07919=1079.560,-94.249,445.798,173.509,19.388,153.355
C07920=1079.565,-94.000,445.787,173.510,19.389,153.355
C07921=1079.571,-93.750,445.778,173.511,19.390,153.355
C07922=1079.577,-93.500,445.767,173.513,19.391,153.355
C07923=1079.583,-93.251,445.757,173.514,19.393,153.355
C07924=1079.590,-93.000,445.746,173.516,19.394,153.355
C07925=1079.596,-92.751,445.736,173.517,19.395,153.355
C07926=1079.602,-92.501,445.725,173.519,19.397,153.355
C07927=1079.608,-92.251,445.716,173.521,19.398,153.355
C07928=1079.614,-92.002,445.705,173.522,19.399,153.355
C07929=1079.620,-91.753,445.695,173.524,19.401,153.355
C07930=1079.625,-91.503,445.685,173.525,19.402,153.355
C07931=1079.631,-91.253,445.674,173.527,19.403,153.355
C07932=1079.638,-91.003,445.664,173.528,19.405,153.355
C07933=1079.644,-90.753,445.653,173.530,19.406,153.355
C07934=1079.650,-90.504,445.643,173.531,19.407,153.355
C07935=1079.656,-90.254,445.632,173.533,19.409,153.355
C07936=1079.662,-90.005,445.622,173.535,19.410,153.355
C07937=1079.668,-89.755,445.612,173.535,19.411,153.355
C07938=1079.674,-89.504,445.601,173.537,19.412,153.355
C07939=1079.680,-89.255,445.590,173.538,19.414,153.355
C07940=1079.686,-89.005,445.580,173.540,19.415,153.355
C07941=1079.692,-88.756,445.570,173.541,19.416,153.355
C07942=1079.698,-88.506,445.559,173.543,19.418,153.355
C07943=1079.704,-88.257,445.550,173.544,19.419,153.355
C07944=1079.710,-88.006,445.538,173.546,19.420,153.355
C07945=1079.716,-87.757,445.527,173.547,19.422,153.355
C07946=1079.722,-87.507,445.518,173.549,19.423,153.355
C07947=1079.728,-87.258,445.507,173.551,19.424,153.355
C07948=1079.735,-87.008,445.497,173.552,19.425,153.355
C07949=1079.741,-86.758,445.486,173.554,19.427,153.355
C07950=1079.746,-86.508,445.475,173.555,19.428,153.355
C07951=1079.753,-86.259,445.465,173.557,19.429,153.354
C07952=1079.759,-86.009,445.454,173.558,19.431,153.355
C07953=1079.765,-85.759,445.444,173.560,19.432,153.355
C07954=1079.771,-85.509,445.433,173.561,19.434,153.355
C07955=1079.777,-85.260,445.422,173.563,19.435,153.355
C07956=1079.783,-85.011,445.412,173.564,19.436,153.354
C07957=1079.789,-84.760,445.402,173.566,19.438,153.354
C07958=1079.795,-84.511,445.391,173.567,19.439,153.355
C07959=1079.802,-84.261,445.380,173.569,19.441,153.355
C07960=1079.807,-84.012,445.370,173.570,19.442,153.354
C07961=1079.813,-83.761,445.359,173.572,19.443,153.354
C07962=1079.820,-83.512,445.349,173.573,19.445,153.354
C07963=1079.826,-83.262,445.338,173.575,19.446,153.355
C07964=1079.832,-83.013,445.328,173.576,19.448,153.355
C07965=1079.838,-82.763,445.316,173.578,19.449,153.355
C07966=1079.844,-82.513,445.306,173.580,19.450,153.354
C07967=1079.850,-82.264,445.296,173.580,19.451,153.355
C07968=1079.857,-82.014,445.285,173.582,19.453,153.355
C07969=1079.863,-81.737,445.273,173.584,19.455,153.355
C07970=1079.870,-81.459,445.261,173.585,19.456,153.355
C07971=1079.877,-81.182,445.249,173.587,19.458,153.355
C07972=1079.884,-80.905,445.237,173.588,19.459,153.355
C07973=1079.890,-80.655,445.227,173.590,19.461,153.355
C07974=1079.895,-80.405,445.216,173.592,19.462,153.355
C07975=1079.902,-80.155,445.205,173.593,19.463,153.355
C07976=1079.908,-79.906,445.194,173.594,19.465,153.355
C07977=1079.914,-79.657,445.184,173.596,19.466,153.355
C07978=1079.920,-79.407,445.173,173.597,19.468,153.355
C07979=1079.926,-79.157,445.161,173.599,19.469,153.355
C07980=1079.932,-78.908,445.151,173.600,19.471,153.355
C07981=1079.938,-78.658,445.140,173.602,19.472,153.355
C07982=1079.945,-78.408,445.129,173.603,19.474,153.355
C07983=1079.950,-78.158,445.119,173.605,19.475,153.355
C07984=1079.956,-77.908,445.108,173.606,19.477,153.355
C07985=1079.961,-77.659,445.097,173.608,19.478,153.355
C07986=1079.968,-77.409,445.086,173.609,19.480,153.355
C07987=1079.974,-77.160,445.076,173.611,19.481,153.355
C07988=1079.980,-76.910,445.065,173.612,19.483,153.355
C07989=1079.986,-76.660,445.053,173.614,19.484,153.355
C07990=1079.992,-76.410,445.043,173.615,19.486,153.355
C07991=1079.998,-76.161,445.032,173.617,19.487,153.355
C07992=1080.004,-75.911,445.021,173.618,19.489,153.355
C07993=1080.010,-75.661,445.010,173.619,19.490,153.355
C07994=1080.016,-75.412,444.999,173.621,19.492,153.355
C07995=1080.022,-75.161,444.988,173.622,19.493,153.355
C07996=1080.029,-74.912,444.977,173.624,19.495,153.355
C07997=1080.034,-74.663,444.966,173.625,19.496,153.355
C07998=1080.041,-74.413,444.955,173.627,19.498,153.355
C07999=1080.046,-74.163,444.944,173.628,19.499,153.355
C08000=1080.052,-73.914,444.933,173.630,19.501,153.355
C08001=1080.058,-73.663,444.922,173.631,19.502,153.355
C08002=1080.064,-73.414,444.911,173.633,19.504,153.355
C08003=1080.070,-73.165,444.900,173.634,19.505,153.355
C08004=1080.076,-72.916,444.889,173.636,19.507,153.355
C08005=1080.082,-72.665,444.878,173.637,19.509,153.356
C08006=1080.087,-72.416,444.866,173.639,19.511,153.355
C08007=1080.093,-72.166,444.855,173.641,19.512,153.356
C08008=1080.099,-71.916,444.844,173.642,19.514,153.356
C08009=1080.105,-71.666,444.833,173.644,19.515,153.356
C08010=1080.111,-71.417,444.822,173.645,19.517,153.356
C08011=1080.117,-71.167,444.811,173.646,19.519,153.356
C08012=1080.123,-70.917,444.800,173.648,19.520,153.356
C08013=1080.129,-70.668,444.789,173.649,19.522,153.356
C08014=1080.135,-70.418,444.777,173.651,19.523,153.356
C08015=1080.141,-70.169,444.766,173.652,19.525,153.356
C08016=1080.146,-69.919,444.755,173.654,19.526,153.356
C08017=1080.152,-69.669,444.744,173.655,19.528,153.356
C08018=1080.158,-69.419,444.733,173.656,19.530,153.356
C08019=1080.164,-69.170,444.722,173.658,19.531,153.356
C08020=1080.170,-68.920,444.710,173.659,19.533,153.356
C08021=1080.176,-68.671,444.699,173.661,19.534,153.356
C08022=1080.183,-68.421,444.688,173.662,19.536,153.356
C08023=1080.188,-68.171,444.677,173.664,19.538,153.356
C08024=1080.193,-67.921,444.665,173.665,19.539,153.356
C08025=1080.200,-67.672,444.653,173.667,19.541,153.356
C08026=1080.206,-67.422,444.643,173.668,19.542,153.356
C08027=1080.211,-67.173,444.632,173.669,19.544,153.357
C08028=1080.218,-66.922,444.620,173.671,19.546,153.357
C08029=1080.224,-66.674,444.609,173.672,19.547,153.357
C08030=1080.229,-66.423,444.597,173.674,19.549,153.357
C08031=1080.235,-66.174,444.586,173.675,19.551,153.357
C08032=1080.242,-65.923,444.575,173.676,19.552,153.357
C08033=1080.248,-65.649,444.562,173.679,19.554,153.357
C08034=1080.254,-65.374,444.550,173.680,19.556,153.357
C08035=1080.261,-65.099,444.538,173.681,19.558,153.357
C08036=1080.268,-64.824,444.524,173.684,19.560,153.357
C08037=1080.273,-64.574,444.514,173.685,19.561,153.357
C08038=1080.280,-64.324,444.502,173.686,19.563,153.357
C08039=1080.286,-64.075,444.491,173.688,19.565,153.357
C08040=1080.291,-63.825,444.480,173.689,19.566,153.357
C08041=1080.298,-63.575,444.469,173.691,19.568,153.358
C08042=1080.303,-63.326,444.456,173.692,19.570,153.358
C08043=1080.309,-63.076,444.445,173.694,19.571,153.358
C08044=1080.315,-62.826,444.434,173.695,19.573,153.358
C08045=1080.322,-62.577,444.422,173.696,19.575,153.358
C08046=1080.328,-62.327,444.411,173.698,19.576,153.358
C08047=1080.333,-62.077,444.400,173.699,19.578,153.358
C08048=1080.339,-61.828,444.388,173.701,19.579,153.358
C08049=1080.346,-61.578,444.377,173.702,19.581,153.358
C08050=1080.352,-61.329,444.365,173.703,19.583,153.358
C08051=1080.357,-61.078,444.353,173.705,19.584,153.358
C08052=1080.363,-60.829,444.342,173.706,19.586,153.358
C08053=1080.370,-60.579,444.331,173.709,19.588,153.358
C08054=1080.375,-60.330,444.320,173.710,19.590,153.358
C08055=1080.382,-60.080,444.308,173.711,19.591,153.358
C08056=1080.387,-59.831,444.296,173.713,19.593,153.358
C08057=1080.393,-59.580,444.285,173.714,19.595,153.358
C08058=1080.399,-59.331,444.273,173.716,19.596,153.359
C08059=1080.406,-59.081,444.262,173.717,19.598,153.359
C08060=1080.411,-58.832,444.250,173.718,19.600,153.359
C08061=1080.417,-58.582,444.239,173.720,19.601,153.359
C08062=1080.423,-58.333,444.227,173.721,19.603,153.359
C08063=1080.430,-58.083,444.216,173.723,19.605,153.359
C08064=1080.436,-57.833,444.203,173.724,19.606,153.359
C08065=1080.441,-57.583,444.192,173.725,19.608,153.359
C08066=1080.448,-57.334,444.180,173.727,19.610,153.359
C08067=1080.454,-57.084,444.170,173.729,19.612,153.359
C08068=1080.460,-56.835,444.157,173.730,19.614,153.359
C08069=1080.465,-56.585,444.146,173.732,19.615,153.359
C08070=1080.472,-56.335,444.134,173.733,19.617,153.359
C08071=1080.478,-56.085,444.122,173.735,19.619,153.360
C08072=1080.484,-55.836,444.111,173.736,19.620,153.360
C08073=1080.490,-55.586,444.100,173.738,19.622,153.360
C08074=1080.496,-55.337,444.088,173.739,19.624,153.360
C08075=1080.502,-55.087,444.075,173.740,19.625,153.360
C08076=1080.508,-54.837,444.064,173.742,19.627,153.360
C08077=1080.514,-54.588,444.053,173.743,19.629,153.360
C08078=1080.520,-54.338,444.041,173.744,19.630,153.360
C08079=1080.526,-54.089,444.029,173.747,19.632,153.360
C08080=1080.533,-53.839,444.017,173.748,19.634,153.360
C08081=1080.539,-53.589,444.006,173.749,19.636,153.360
C08082=1080.544,-53.340,443.994,173.751,19.637,153.360
C08083=1080.551,-53.090,443.982,173.752,19.639,153.360
C08084=1080.557,-52.840,443.971,173.754,19.641,153.360
C08085=1080.563,-52.591,443.958,173.755,19.643,153.361
C08086=1080.569,-52.341,443.947,173.756,19.644,153.361
C08087=1080.576,-52.091,443.935,173.758,19.646,153.361
C08088=1080.581,-51.842,443.923,173.759,19.648,153.361
C08089=1080.587,-51.592,443.912,173.761,19.649,153.361
C08090=1080.594,-51.342,443.900,173.763,19.651,153.361
C08091=1080.599,-51.093,443.888,173.764,19.653,153.361
C08092=1080.606,-50.843,443.876,173.766,19.655,153.361
C08093=1080.612,-50.593,443.864,173.767,19.657,153.361
C08094=1080.618,-50.344,443.852,173.768,19.658,153.361
C08095=1080.624,-50.094,443.841,173.770,19.660,153.361
C08096=1080.629,-49.845,443.829,173.771,19.662,153.361
C08097=1080.636,-49.571,443.815,173.772,19.664,153.362
C08098=1080.643,-49.296,443.802,173.774,19.666,153.362
C08099=1080.649,-49.023,443.789,173.776,19.668,153.362
C08100=1080.656,-48.749,443.775,173.777,19.670,153.362
C08101=1080.661,-48.500,443.765,173.779,19.672,153.362
C08102=1080.667,-48.250,443.752,173.781,19.674,153.362
C08103=1080.673,-48.001,443.740,173.782,19.676,153.362
C08104=1080.679,-47.751,443.728,173.783,19.677,153.362
C08105=1080.689,-47.335,443.708,173.785,19.680,153.363
C08106=1080.699,-46.921,443.689,173.788,19.683,153.363
C08107=1080.709,-46.506,443.668,173.790,19.686,153.363
C08108=1080.718,-46.090,443.648,173.793,19.689,153.363
C08109=1080.725,-45.841,443.636,173.794,19.691,153.363
C08110=1080.730,-45.591,443.624,173.796,19.694,153.363
C08111=1080.736,-45.342,443.611,173.797,19.695,153.363
C08112=1080.742,-45.093,443.600,173.798,19.697,153.364
C08113=1080.748,-44.843,443.587,173.800,19.699,153.364
C08114=1080.754,-44.592,443.575,173.802,19.701,153.364
C08115=1080.760,-44.343,443.564,173.803,19.703,153.364
C08116=1080.766,-44.094,443.551,173.805,19.705,153.364
C08117=1080.772,-43.844,443.539,173.806,19.707,153.364
C08118=1080.778,-43.595,443.527,173.807,19.708,153.364
C08119=1080.784,-43.345,443.514,173.809,19.710,153.364
C08120=1080.790,-43.095,443.502,173.810,19.712,153.364
C08121=1080.796,-42.846,443.490,173.811,19.714,153.364
C08122=1080.801,-42.596,443.478,173.813,19.716,153.365
C08123=1080.808,-42.346,443.466,173.815,19.718,153.365
C08124=1080.814,-42.096,443.454,173.816,19.720,153.365
C08125=1080.819,-41.847,443.442,173.818,19.721,153.365
C08126=1080.826,-41.597,443.430,173.819,19.723,153.365
C08127=1080.832,-41.348,443.417,173.820,19.725,153.365
C08128=1080.838,-41.098,443.405,173.822,19.727,153.365
C08129=1080.843,-40.848,443.392,173.823,19.729,153.365
C08130=1080.850,-40.599,443.380,173.825,19.731,153.365
C08131=1080.855,-40.349,443.368,173.826,19.733,153.365
C08132=1080.861,-40.099,443.355,173.828,19.735,153.366
C08133=1080.867,-39.850,443.344,173.829,19.736,153.366
C08134=1080.873,-39.600,443.331,173.830,19.738,153.366
C08135=1080.879,-39.351,443.319,173.832,19.740,153.366
C08136=1080.886,-39.101,443.307,173.833,19.742,153.366
C08137=1080.891,-38.852,443.295,173.835,19.744,153.366
C08138=1080.897,-38.602,443.282,173.837,19.746,153.366
C08139=1080.903,-38.352,443.269,173.838,19.748,153.366
C08140=1080.910,-38.102,443.257,173.839,19.750,153.367
C08141=1080.915,-37.853,443.245,173.841,19.751,153.367
C08142=1080.921,-37.603,443.233,173.842,19.753,153.367
C08143=1080.927,-37.353,443.220,173.843,19.755,153.367
C08144=1080.933,-37.104,443.208,173.846,19.757,153.367
C08145=1080.938,-36.854,443.195,173.847,19.759,153.367
C08146=1080.944,-36.605,443.182,173.848,19.761,153.367
C08147=1080.950,-36.355,443.170,173.849,19.763,153.367
C08148=1080.957,-36.106,443.158,173.851,19.765,153.367
C08149=1080.962,-35.857,443.145,173.852,19.767,153.368
C08150=1080.968,-35.607,443.133,173.853,19.769,153.368
C08151=1080.974,-35.357,443.120,173.855,19.771,153.368
C08152=1080.980,-35.107,443.108,173.857,19.773,153.368
C08153=1080.986,-34.857,443.095,173.858,19.775,153.368
C08154=1080.991,-34.608,443.083,173.859,19.777,153.368
C08155=1080.997,-34.359,443.070,173.861,19.778,153.368
C08156=1081.003,-34.109,443.057,173.862,19.780,153.369
C08157=1081.012,-33.751,443.040,173.864,19.783,153.369
C08158=1081.020,-33.394,443.022,173.867,19.786,153.369
C08159=1081.029,-33.035,443.003,173.869,19.789,153.369
C08160=1081.037,-32.678,442.986,173.871,19.792,153.369
C08161=1081.043,-32.428,442.973,173.872,19.794,153.369
C08162=1081.049,-32.178,442.961,173.873,19.796,153.370
C08163=1081.055,-31.930,442.948,173.875,19.797,153.370
C08164=1081.061,-31.680,442.935,173.876,19.799,153.370
C08165=1081.067,-31.430,442.923,173.877,19.801,153.370
C08166=1081.072,-31.180,442.910,173.879,19.804,153.370
C08167=1081.079,-30.931,442.897,173.881,19.805,153.370
C08168=1081.085,-30.681,442.884,173.882,19.807,153.370
C08169=1081.090,-30.431,442.872,173.883,19.809,153.370
C08170=1081.096,-30.182,442.859,173.885,19.811,153.371
C08171=1081.102,-29.933,442.846,173.886,19.813,153.371
C08172=1081.109,-29.683,442.834,173.888,19.815,153.371
C08173=1081.115,-29.433,442.822,173.890,19.817,153.371
C08174=1081.121,-29.184,442.808,173.891,19.819,153.371
C08175=1081.127,-28.934,442.796,173.892,19.821,153.371
C08176=1081.133,-28.684,442.783,173.894,19.823,153.371
C08177=1081.138,-28.434,442.771,173.895,19.825,153.371
C08178=1081.145,-28.185,442.757,173.897,19.827,153.372
C08179=1081.150,-27.936,442.745,173.898,19.829,153.372
C08180=1081.156,-27.686,442.733,173.900,19.831,153.372
C08181=1081.162,-27.437,442.719,173.901,19.833,153.372
C08182=1081.168,-27.187,442.707,173.902,19.835,153.372
C08183=1081.174,-26.937,442.694,173.904,19.836,153.372
C08184=1081.180,-26.688,442.681,173.906,19.839,153.372
C08185=1081.186,-26.438,442.668,173.907,19.841,153.372
C08186=1081.192,-26.188,442.655,173.908,19.843,153.373
C08187=1081.197,-25.938,442.642,173.910,19.845,153.373
C08188=1081.203,-25.689,442.630,173.911,19.847,153.373
C08189=1081.209,-25.440,442.617,173.912,19.848,153.373
C08190=1081.215,-25.190,442.604,173.914,19.851,153.373
C08191=1081.221,-24.941,442.591,173.916,19.853,153.373
C08192=1081.226,-24.690,442.578,173.917,19.855,153.374
C08193=1081.232,-24.441,442.564,173.918,19.857,153.374
C08194=1081.238,-24.191,442.552,173.919,19.859,153.374
C08195=1081.244,-23.941,442.539,173.921,19.861,153.374
C08196=1081.251,-23.692,442.526,173.923,19.863,153.374
C08197=1081.256,-23.442,442.513,173.924,19.865,153.374
C08198=1081.262,-23.193,442.500,173.925,19.867,153.374
C08199=1081.267,-22.943,442.487,173.927,19.869,153.375
C08200=1081.273,-22.694,442.474,173.928,19.871,153.375
C08201=1081.279,-22.444,442.462,173.930,19.873,153.375
C08202=1081.285,-22.195,442.448,173.931,19.875,153.375
C08203=1081.291,-21.945,442.435,173.933,19.877,153.375
C08204=1081.297,-21.696,442.422,173.934,19.879,153.375
C08205=1081.303,-21.446,442.409,173.935,19.881,153.375
C08206=1081.309,-21.196,442.396,173.937,19.883,153.376
C08207=1081.314,-20.946,442.383,173.939,19.885,153.376
C08208=1081.320,-20.697,442.370,173.940,19.887,153.376
C08209=1081.327,-20.448,442.356,173.941,19.889,153.376
C08210=1081.333,-20.198,442.344,173.942,19.891,153.376
C08211=1081.339,-19.949,442.331,173.945,19.894,153.376
C08212=1081.344,-19.698,442.317,173.946,19.895,153.376
C08213=1081.350,-19.449,442.304,173.947,19.897,153.377
C08214=1081.356,-19.199,442.292,173.949,19.899,153.377
C08215=1081.362,-18.950,442.278,173.950,19.901,153.377
C08216=1081.368,-18.700,442.264,173.951,19.903,153.377
C08217=1081.374,-18.451,442.252,173.953,19.906,153.377
C08218=1081.380,-18.201,442.239,173.954,19.908,153.377
C08219=1081.386,-17.951,442.226,173.956,19.910,153.378
C08220=1081.391,-17.702,442.212,173.957,19.911,153.378
C08221=1081.398,-17.428,442.198,173.959,19.914,153.378
C08222=1081.405,-17.154,442.183,173.960,19.917,153.378
C08223=1081.411,-16.879,442.169,173.962,19.919,153.378
C08224=1081.418,-16.605,442.155,173.964,19.921,153.378
C08225=1081.424,-16.355,442.141,173.965,19.923,153.378
C08226=1081.430,-16.106,442.127,173.966,19.924,153.378
C08227=1081.436,-15.856,442.115,173.968,19.927,153.379
C08228=1081.442,-15.607,442.102,173.970,19.929,153.379
C08229=1081.447,-15.357,442.088,173.971,19.931,153.379
C08230=1081.453,-15.107,442.075,173.972,19.933,153.379
C08231=1081.459,-14.858,442.062,173.974,19.935,153.379
C08232=1081.465,-14.608,442.048,173.975,19.937,153.379
C08233=1081.471,-14.359,442.035,173.977,19.940,153.380
C08234=1081.476,-14.109,442.022,173.978,19.942,153.380
C08235=1081.482,-13.860,442.008,173.980,19.944,153.380
C08236=1081.488,-13.610,441.995,173.981,19.946,153.380
C08237=1081.494,-13.361,441.981,173.983,19.948,153.380
C08238=1081.500,-13.111,441.969,173.984,19.950,153.380
C08239=1081.505,-12.861,441.955,173.985,19.952,153.381
C08240=1081.512,-12.612,441.942,173.987,19.954,153.381
C08241=1081.517,-12.363,441.928,173.988,19.956,153.381
C08242=1081.523,-12.113,441.914,173.990,19.959,153.381
C08243=1081.529,-11.863,441.901,173.991,19.961,153.381
C08244=1081.535,-11.614,441.888,173.993,19.963,153.381
C08245=1081.540,-11.364,441.874,173.994,19.965,153.382
C08246=1081.546,-11.115,441.861,173.995,19.966,153.382
C08247=1081.553,-10.865,441.847,173.997,19.969,153.382
C08248=1081.558,-10.615,441.834,173.999,19.971,153.382
C08249=1081.564,-10.365,441.820,174.000,19.973,153.382
C08250=1081.570,-10.116,441.807,174.001,19.975,153.382
C08251=1081.576,-9.866,441.793,174.002,19.977,153.382
C08252=1081.582,-9.617,441.780,174.005,19.979,153.383
C08253=1081.587,-9.368,441.766,174.006,19.981,153.383
C08254=1081.594,-9.118,441.753,174.007,19.983,153.383
C08255=1081.599,-8.869,441.739,174.008,19.985,153.383
C08256=1081.605,-8.619,441.726,174.010,19.988,153.383
C08257=1081.611,-8.369,441.712,174.012,19.990,153.383
C08258=1081.617,-8.119,441.699,174.013,19.992,153.384
C08259=1081.623,-7.870,441.685,174.014,19.994,153.384
C08260=1081.629,-7.620,441.672,174.016,19.996,153.384
C08261=1081.634,-7.371,441.658,174.018,19.998,153.384
C08262=1081.641,-7.122,441.644,174.019,20.000,153.384
C08263=1081.646,-6.872,441.631,174.020,20.002,153.384
C08264=1081.653,-6.622,441.617,174.021,20.004,153.385
C08265=1081.658,-6.372,441.603,174.024,20.007,153.385
C08266=1081.664,-6.123,441.589,174.025,20.009,153.385
C08267=1081.670,-5.874,441.576,174.026,20.011,153.385
C08268=1081.676,-5.624,441.562,174.027,20.013,153.385
C08269=1081.682,-5.375,441.549,174.029,20.015,153.385
C08270=1081.688,-5.125,441.535,174.031,20.017,153.386
C08271=1081.694,-4.875,441.521,174.032,20.019,153.386
C08272=1081.699,-4.626,441.507,174.033,20.021,153.386
C08273=1081.706,-4.376,441.494,174.034,20.023,153.386
C08274=1081.711,-4.127,441.480,174.037,20.026,153.386
C08275=1081.717,-3.877,441.466,174.038,20.028,153.386
C08276=1081.723,-3.627,441.453,174.039,20.030,153.387
C08277=1081.729,-3.378,441.439,174.041,20.031,153.387
C08278=1081.735,-3.128,441.426,174.042,20.034,153.387
C08279=1081.741,-2.879,441.412,174.044,20.036,153.387
C08280=1081.746,-2.629,441.398,174.045,20.038,153.387
C08281=1081.752,-2.379,441.384,174.046,20.040,153.387
C08282=1081.758,-2.129,441.370,174.048,20.042,153.388
C08283=1081.764,-1.881,441.356,174.050,20.045,153.388
C08284=1081.770,-1.631,441.342,174.051,20.047,153.388
C08285=1081.776,-1.355,441.326,174.052,20.049,153.388
C08286=1081.782,-1.079,441.312,174.054,20.052,153.388
C08287=1081.788,-0.803,441.296,174.055,20.054,153.388
C08288=1081.795,-0.528,441.281,174.058,20.056,153.389
C08289=1081.800,-0.278,441.267,174.059,20.058,153.389
C08290=1081.806,-0.029,441.253,174.060,20.060,153.389
C08291=1081.812,0.221,441.238,174.062,20.062,153.389
C08292=1081.818,0.471,441.224,174.063,20.064,153.389
C08293=1081.824,0.720,441.211,174.064,20.067,153.390
C08294=1081.829,0.970,441.197,174.066,20.069,153.390
C08295=1081.835,1.219,441.183,174.067,20.071,153.390
C08296=1081.841,1.469,441.169,174.069,20.074,153.390
C08297=1081.847,1.718,441.155,174.070,20.076,153.390
C08298=1081.852,1.968,441.141,174.072,20.078,153.390
C08299=1081.859,2.217,441.128,174.073,20.080,153.391
C08300=1081.865,2.467,441.113,174.075,20.082,153.391
C08301=1081.870,2.716,441.099,174.076,20.084,153.391
C08302=1081.876,2.966,441.085,174.078,20.086,153.391
C08303=1081.881,3.216,441.071,174.079,20.088,153.391
C08304=1081.887,3.465,441.057,174.081,20.090,153.391
C08305=1081.894,3.714,441.043,174.082,20.092,153.391
C08306=1081.899,3.964,441.029,174.083,20.094,153.392
C08307=1081.905,4.214,441.015,174.085,20.097,153.392
C08308=1081.911,4.463,441.000,174.087,20.099,153.392
C08309=1081.917,4.713,440.986,174.088,20.101,153.392
C08310=1081.922,4.962,440.972,174.089,20.103,153.392
C08311=1081.928,5.212,440.959,174.090,20.105,153.393
C08312=1081.934,5.462,440.944,174.093,20.108,153.393
C08313=1081.940,5.711,440.930,174.094,20.110,153.393
C08314=1081.946,5.960,440.916,174.095,20.112,153.393
C08315=1081.952,6.209,440.902,174.096,20.114,153.393
C08316=1081.958,6.460,440.888,174.099,20.116,153.393
C08317=1081.963,6.709,440.873,174.100,20.118,153.394
C08318=1081.969,6.958,440.859,174.101,20.120,153.394
C08319=1081.975,7.209,440.845,174.102,20.122,153.394
C08320=1081.981,7.457,440.830,174.104,20.125,153.394
C08321=1081.986,7.707,440.817,174.106,20.127,153.394
C08322=1081.992,7.957,440.802,174.107,20.129,153.394
C08323=1081.998,8.206,440.788,174.108,20.131,153.395
C08324=1082.004,8.456,440.774,174.110,20.133,153.395
C08325=1082.011,8.705,440.759,174.112,20.135,153.395
C08326=1082.016,8.955,440.746,174.113,20.137,153.395
C08327=1082.022,9.204,440.731,174.115,20.140,153.395
C08328=1082.028,9.454,440.717,174.116,20.142,153.396
C08329=1082.033,9.704,440.703,174.117,20.144,153.396
C08330=1082.039,9.953,440.688,174.119,20.146,153.396
C08331=1082.045,10.203,440.674,174.121,20.149,153.396
C08332=1082.051,10.452,440.660,174.122,20.151,153.396
C08333=1082.057,10.702,440.645,174.123,20.153,153.396
C08334=1082.063,10.951,440.631,174.125,20.155,153.397
C08335=1082.068,11.201,440.617,174.127,20.157,153.397
C08336=1082.075,11.450,440.602,174.128,20.159,153.397
C08337=1082.080,11.700,440.588,174.129,20.161,153.397
C08338=1082.087,11.949,440.573,174.130,20.163,153.397
C08339=1082.092,12.199,440.559,174.133,20.166,153.397
C08340=1082.098,12.448,440.545,174.134,20.168,153.397
C08341=1082.104,12.698,440.530,174.135,20.170,153.398
C08342=1082.110,12.947,440.516,174.136,20.172,153.398
C08343=1082.116,13.197,440.501,174.139,20.174,153.398
C08344=1082.122,13.446,440.487,174.140,20.176,153.398
C08345=1082.128,13.695,440.473,174.141,20.178,153.398
C08346=1082.134,13.945,440.459,174.143,20.181,153.398
C08347=1082.140,14.194,440.444,174.145,20.183,153.399
C08348=1082.146,14.444,440.429,174.146,20.185,153.399
C08349=1082.152,14.722,440.413,174.148,20.187,153.399
C08350=1082.159,15.000,440.397,174.149,20.190,153.399
C08351=1082.165,15.278,440.381,174.151,20.192,153.399
C08352=1082.172,15.555,440.364,174.152,20.194,153.400
C08353=1082.177,15.805,440.350,174.154,20.196,153.400
C08354=1082.184,16.055,440.335,174.156,20.199,153.400
C08355=1082.189,16.304,440.322,174.157,20.201,153.400
C08356=1082.195,16.554,440.306,174.158,20.203,153.400
C08357=1082.200,16.803,440.291,174.160,20.206,153.400
C08358=1082.206,17.053,440.278,174.161,20.208,153.401
C08359=1082.212,17.302,440.263,174.163,20.210,153.401
C08360=1082.218,17.551,440.248,174.164,20.212,153.401
C08361=1082.224,17.801,440.233,174.166,20.214,153.401
C08362=1082.229,18.051,440.219,174.167,20.216,153.401
C08363=1082.236,18.300,440.204,174.169,20.218,153.401
C08364=1082.241,18.549,440.189,174.171,20.220,153.402
C08365=1082.247,18.800,440.175,174.172,20.222,153.402
C08366=1082.253,19.049,440.160,174.173,20.225,153.402
C08367=1082.258,19.298,440.145,174.174,20.227,153.402
C08368=1082.265,19.548,440.130,174.177,20.229,153.402
C08369=1082.270,19.797,440.116,174.178,20.231,153.403
C08370=1082.277,20.047,440.101,174.179,20.233,153.403
C08371=1082.282,20.296,440.086,174.181,20.236,153.403
C08372=1082.288,20.546,440.071,174.183,20.238,153.403
C08373=1082.294,20.795,440.057,174.184,20.240,153.403
C08374=1082.300,21.045,440.042,174.185,20.242,153.403
C08375=1082.305,21.294,440.027,174.187,20.244,153.404
C08376=1082.311,21.544,440.012,174.188,20.246,153.404
C08377=1082.317,21.793,439.998,174.190,20.248,153.404
C08378=1082.323,22.043,439.982,174.192,20.251,153.404
C08379=1082.328,22.292,439.968,174.193,20.253,153.404
C08380=1082.334,22.542,439.953,174.194,20.255,153.405
C08381=1082.340,22.791,439.938,174.195,20.257,153.405
C08382=1082.346,23.041,439.923,174.198,20.260,153.405
C08383=1082.352,23.290,439.909,174.199,20.262,153.405
C08384=1082.357,23.540,439.893,174.200,20.264,153.405
C08385=1082.363,23.789,439.879,174.202,20.266,153.405
C08386=1082.370,24.039,439.864,174.204,20.268,153.405
C08387=1082.374,24.288,439.849,174.205,20.270,153.406
C08388=1082.381,24.538,439.834,174.207,20.273,153.406
C08389=1082.386,24.787,439.820,174.208,20.275,153.406
C08390=1082.392,25.037,439.804,174.209,20.277,153.406
C08391=1082.398,25.286,439.789,174.211,20.279,153.406
C08392=1082.403,25.536,439.774,174.213,20.282,153.407
C08393=1082.409,25.785,439.759,174.214,20.284,153.407
C08394=1082.416,26.035,439.744,174.215,20.286,153.407
C08395=1082.421,26.284,439.729,174.217,20.288,153.407
C08396=1082.427,26.533,439.714,174.219,20.290,153.407
C08397=1082.433,26.783,439.699,174.220,20.292,153.407
C08398=1082.439,27.032,439.684,174.222,20.295,153.408
C08399=1082.445,27.282,439.669,174.223,20.297,153.408
C08400=1082.450,27.531,439.654,174.225,20.299,153.408
C08401=1082.456,27.781,439.639,174.226,20.300,153.408
C08402=1082.461,28.030,439.624,174.228,20.303,153.408
C08403=1082.468,28.280,439.609,174.229,20.305,153.408
C08404=1082.474,28.530,439.594,174.230,20.307,153.409
C08405=1082.479,28.779,439.579,174.233,20.310,153.409
C08406=1082.486,29.028,439.564,174.234,20.312,153.409
C08407=1082.491,29.278,439.549,174.235,20.314,153.409
C08408=1082.497,29.527,439.534,174.237,20.316,153.409
C08409=1082.502,29.777,439.519,174.239,20.318,153.409
C08410=1082.508,30.026,439.504,174.240,20.320,153.410
C08411=1082.514,30.276,439.487,174.242,20.323,153.410
C08412=1082.519,30.525,439.472,174.243,20.325,153.410
C08413=1082.526,30.804,439.455,174.244,20.327,153.410
C08414=1082.533,31.084,439.438,174.246,20.330,153.410
C08415=1082.539,31.363,439.422,174.249,20.332,153.411
C08416=1082.545,31.643,439.405,174.250,20.335,153.411
C08417=1082.551,31.891,439.389,174.252,20.337,153.411
C08418=1082.557,32.141,439.374,174.253,20.339,153.411
C08419=1082.563,32.390,439.359,174.254,20.341,153.411
C08420=1082.569,32.640,439.344,174.256,20.344,153.411
C08421=1082.574,32.890,439.328,174.258,20.346,153.412
C08422=1082.580,33.139,439.313,174.259,20.348,153.412
C08423=1082.586,33.388,439.297,174.260,20.350,153.412
C08424=1082.592,33.637,439.283,174.262,20.352,153.412
C08425=1082.597,33.887,439.267,174.264,20.354,153.412
C08426=1082.603,34.137,439.252,174.265,20.356,153.413
C08427=1082.609,34.386,439.237,174.267,20.359,153.413
C08428=1082.615,34.635,439.221,174.268,20.361,153.413
C08429=1082.621,34.885,439.206,174.269,20.363,153.413
C08430=1082.626,35.134,439.191,174.272,20.365,153.413
C08431=1082.632,35.384,439.175,174.273,20.367,153.413
C08432=1082.638,35.633,439.159,174.274,20.369,153.414
C08433=1082.644,35.883,439.144,174.276,20.372,153.414
C08434=1082.649,36.133,439.129,174.278,20.374,153.414
C08435=1082.656,36.382,439.114,174.279,20.376,153.414
C08436=1082.661,36.631,439.098,174.281,20.378,153.414
C08437=1082.667,36.881,439.083,174.282,20.380,153.414
C08438=1082.673,37.131,439.067,174.284,20.382,153.415
C08439=1082.679,37.380,439.051,174.286,20.385,153.415
C08440=1082.685,37.629,439.037,174.287,20.387,153.415
C08441=1082.690,37.879,439.021,174.288,20.389,153.415
C08442=1082.696,38.128,439.005,174.290,20.391,153.415
C08443=1082.701,38.377,438.990,174.292,20.393,153.415
C08444=1082.708,38.627,438.975,174.293,20.395,153.416
C08445=1082.714,38.876,438.958,174.295,20.398,153.416
C08446=1082.719,39.126,438.943,174.296,20.400,153.416
C08447=1082.725,39.375,438.927,174.297,20.402,153.416
C08448=1082.730,39.625,438.911,174.300,20.405,153.416
C08449=1082.736,39.874,438.897,174.301,20.407,153.416
C08450=1082.742,40.123,438.881,174.302,20.409,153.417
C08451=1082.748,40.373,438.865,174.304,20.411,153.417
C08452=1082.753,40.622,438.849,174.306,20.413,153.417
C08453=1082.759,40.872,438.834,174.307,20.415,153.417
C08454=1082.765,41.122,438.819,174.309,20.417,153.417
C08455=1082.771,41.371,438.802,174.310,20.419,153.417
C08456=1082.776,41.620,438.787,174.312,20.422,153.418
C08457=1082.782,41.869,438.771,174.314,20.424,153.418
C08458=1082.788,42.119,438.755,174.315,20.426,153.418
C08459=1082.794,42.369,438.739,174.317,20.428,153.418
C08460=1082.799,42.618,438.725,174.318,20.430,153.418
C08461=1082.805,42.867,438.708,174.320,20.433,153.419
C08462=1082.811,43.117,438.693,174.322,20.435,153.419
C08463=1082.817,43.366,438.677,174.323,20.437,153.419
C08464=1082.822,43.616,438.661,174.324,20.439,153.419
C08465=1082.828,43.865,438.645,174.326,20.442,153.419
C08466=1082.834,44.115,438.630,174.328,20.444,153.419
C08467=1082.840,44.364,438.613,174.329,20.446,153.420
C08468=1082.845,44.614,438.598,174.331,20.448,153.420
C08469=1082.851,44.863,438.582,174.332,20.450,153.420
C08470=1082.856,45.113,438.566,174.334,20.452,153.420
C08471=1082.862,45.362,438.550,174.336,20.454,153.420
C08472=1082.867,45.611,438.534,174.337,20.456,153.420
C08473=1082.873,45.861,438.519,174.339,20.459,153.421
C08474=1082.879,46.110,438.502,174.340,20.461,153.421
C08475=1082.884,46.360,438.487,174.342,20.463,153.421
C08476=1082.890,46.609,438.471,174.344,20.466,153.421
C08477=1082.896,46.888,438.454,174.345,20.468,153.421
C08478=1082.903,47.167,438.435,174.347,20.471,153.422
C08479=1082.909,47.447,438.418,174.349,20.473,153.422
C08480=1082.915,47.725,438.400,174.350,20.475,153.422
C08481=1082.921,47.975,438.384,174.353,20.478,153.422
C08482=1082.927,48.225,438.368,174.354,20.480,153.422
C08483=1082.932,48.474,438.351,174.355,20.482,153.422
C08484=1082.938,48.724,438.335,174.357,20.484,153.423
C08485=1082.943,48.973,438.320,174.359,20.486,153.423
C08486=1082.949,49.222,438.304,174.360,20.489,153.423
C08487=1082.955,49.472,438.287,174.362,20.491,153.423
C08488=1082.961,49.722,438.272,174.363,20.493,153.423
C08489=1082.967,49.971,438.256,174.365,20.495,153.423
C08490=1082.972,50.220,438.240,174.367,20.497,153.424
C08491=1082.978,50.470,438.224,174.368,20.499,153.424
C08492=1082.984,50.719,438.208,174.370,20.502,153.424
C08493=1082.990,50.968,438.192,174.371,20.504,153.424
C08494=1082.996,51.218,438.175,174.373,20.506,153.424
C08495=1083.001,51.467,438.158,174.375,20.508,153.424
C08496=1083.006,51.717,438.143,174.376,20.510,153.425
C08497=1083.012,51.966,438.127,174.378,20.513,153.425
C08498=1083.018,52.215,438.111,174.379,20.515,153.425
C08499=1083.024,52.465,438.095,174.381,20.517,153.425
C08500=1083.029,52.715,438.079,174.383,20.519,153.425
C08501=1083.035,52.964,438.063,174.384,20.521,153.425
C08502=1083.041,53.213,438.046,174.385,20.523,153.426
C08503=1083.046,53.463,438.030,174.388,20.525,153.426
C08504=1083.052,53.712,438.014,174.389,20.527,153.426
C08505=1083.058,53.961,437.997,174.391,20.530,153.426
C08506=1083.063,54.211,437.982,174.392,20.532,153.426
C08507=1083.069,54.460,437.966,174.394,20.534,153.426
C08508=1083.075,54.710,437.949,174.396,20.536,153.427
C08509=1083.081,54.959,437.933,174.397,20.538,153.427
C08510=1083.086,55.209,437.916,174.398,20.540,153.427
C08511=1083.092,55.458,437.900,174.401,20.543,153.427
C08512=1083.098,55.707,437.884,174.402,20.545,153.427
C08513=1083.104,55.957,437.868,174.404,20.547,153.427
C08514=1083.110,56.206,437.851,174.405,20.549,153.428
C08515=1083.116,56.455,437.835,174.407,20.551,153.428
C08516=1083.121,56.704,437.819,174.409,20.553,153.428
C08517=1083.127,56.954,437.803,174.410,20.555,153.428
C08518=1083.132,57.204,437.787,174.412,20.557,153.428
C08519=1083.138,57.453,437.770,174.414,20.559,153.428
C08520=1083.144,57.702,437.754,174.415,20.561,153.428
C08521=1083.150,57.952,437.738,174.417,20.564,153.428
C08522=1083.156,58.201,437.721,174.418,20.566,153.429
C08523=1083.161,58.451,437.705,174.421,20.568,153.429
C08524=1083.167,58.700,437.689,174.422,20.570,153.429
C08525=1083.173,58.949,437.672,174.423,20.572,153.429
C08526=1083.179,59.199,437.656,174.425,20.575,153.429
C08527=1083.185,59.448,437.639,174.427,20.577,153.429
C08528=1083.190,59.698,437.623,174.429,20.579,153.430
C08529=1083.197,59.947,437.606,174.430,20.581,153.430
C08530=1083.203,60.196,437.590,174.432,20.583,153.430
C08531=1083.208,60.446,437.573,174.434,20.585,153.430
C08532=1083.214,60.695,437.557,174.435,20.587,153.430
C08533=1083.220,60.944,437.540,174.437,20.589,153.430
C08534=1083.226,61.194,437.524,174.438,20.591,153.430
C08535=1083.232,61.443,437.508,174.440,20.593,153.431
C08536=1083.237,61.693,437.491,174.442,20.596,153.431
C08537=1083.243,61.942,437.475,174.443,20.597,153.431
C08538=1083.249,62.192,437.458,174.446,20.600,153.431
C08539=1083.255,62.441,437.442,174.447,20.602,153.431
C08540=1083.261,62.690,437.424,174.448,20.604,153.431
C08541=1083.267,62.969,437.406,174.450,20.606,153.431
C08542=1083.274,63.248,437.388,174.452,20.609,153.432
C08543=1083.281,63.528,437.370,174.454,20.610,153.432
C08544=1083.287,63.807,437.351,174.456,20.613,153.432
C08545=1083.293,64.055,437.334,174.458,20.615,153.432
C08546=1083.299,64.305,437.318,174.459,20.617,153.432
C08547=1083.304,64.554,437.301,174.461,20.619,153.432
C08548=1083.310,64.804,437.285,174.463,20.622,153.433
C08549=1083.315,65.053,437.268,174.464,20.623,153.433
C08550=1083.322,65.302,437.251,174.466,20.626,153.433
C08551=1083.328,65.552,437.235,174.468,20.628,153.433
C08552=1083.333,65.801,437.218,174.469,20.630,153.433
C08553=1083.339,66.051,437.201,174.471,20.632,153.433
C08554=1083.344,66.300,437.184,174.473,20.634,153.433
C08555=1083.351,66.550,437.167,174.475,20.636,153.434
C08556=1083.356,66.799,437.150,174.476,20.638,153.434
C08557=1083.362,67.049,437.134,174.478,20.641,153.434
C08558=1083.368,67.298,437.117,174.480,20.642,153.434
C08559=1083.373,67.547,437.100,174.481,20.644,153.434
C08560=1083.379,67.797,437.083,174.483,20.647,153.434
C08561=1083.385,68.045,437.066,174.484,20.649,153.434
C08562=1083.390,68.295,437.050,174.487,20.651,153.434
C08563=1083.396,68.544,437.033,174.488,20.653,153.435
C08564=1083.402,68.793,437.016,174.489,20.655,153.435
C08565=1083.408,69.043,437.000,174.491,20.658,153.435
C08566=1083.413,69.293,436.983,174.493,20.659,153.435
C08567=1083.420,69.542,436.965,174.495,20.661,153.435
C08568=1083.425,69.792,436.948,174.496,20.663,153.435
C08569=1083.431,70.041,436.932,174.498,20.666,153.435
C08570=1083.436,70.290,436.915,174.500,20.668,153.436
C08571=1083.442,70.540,436.898,174.501,20.670,153.436
C08572=1083.448,70.788,436.881,174.503,20.672,153.436
C08573=1083.453,71.038,436.864,174.505,20.674,153.436
C08574=1083.458,71.288,436.847,174.507,20.676,153.436
C08575=1083.464,71.536,436.830,174.508,20.678,153.436
C08576=1083.470,71.787,436.813,174.510,20.680,153.436
C08577=1083.477,72.036,436.796,174.512,20.682,153.437
C08578=1083.482,72.285,436.779,174.514,20.685,153.437
C08579=1083.487,72.534,436.762,174.515,20.687,153.437
C08580=1083.493,72.784,436.745,174.517,20.688,153.437
C08581=1083.499,73.033,436.728,174.519,20.691,153.437
C08582=1083.504,73.282,436.711,174.520,20.693,153.437
C08583=1083.510,73.531,436.694,174.522,20.695,153.437
C08584=1083.516,73.781,436.677,174.524,20.697,153.438
C08585=1083.522,74.030,436.659,174.526,20.700,153.438
C08586=1083.527,74.280,436.643,174.527,20.701,153.438
C08587=1083.533,74.529,436.625,174.529,20.703,153.438
C08588=1083.538,74.778,436.608,174.531,20.705,153.438
C08589=1083.544,75.027,436.591,174.532,20.707,153.438
C08590=1083.550,75.278,436.574,174.534,20.710,153.438
C08591=1083.556,75.527,436.557,174.535,20.712,153.439
C08592=1083.561,75.776,436.540,174.538,20.714,153.439
C08593=1083.567,76.025,436.523,174.539,20.716,153.439
C08594=1083.573,76.274,436.505,174.541,20.718,153.439
C08595=1083.579,76.524,436.488,174.543,20.720,153.439
C08596=1083.584,76.773,436.471,174.545,20.722,153.439
C08597=1083.590,77.023,436.454,174.546,20.724,153.439
C08598=1083.596,77.272,436.437,174.548,20.726,153.439
C08599=1083.601,77.521,436.419,174.550,20.728,153.440
C08600=1083.608,77.771,436.403,174.551,20.730,153.440
C08601=1083.613,78.020,436.385,174.553,20.732,153.440
C08602=1083.619,78.269,436.367,174.555,20.734,153.440
C08603=1083.624,78.519,436.351,174.557,20.737,153.440
C08604=1083.630,78.768,436.333,174.558,20.739,153.440
C08605=1083.636,79.047,436.313,174.560,20.741,153.440
C08606=1083.643,79.325,436.294,174.563,20.743,153.441
C08607=1083.649,79.605,436.275,174.564,20.745,153.441
C08608=1083.655,79.883,436.256,174.566,20.748,153.441
C08609=1083.662,80.133,436.238,174.568,20.750,153.441
C08610=1083.667,80.382,436.220,174.570,20.752,153.441
C08611=1083.672,80.632,436.203,174.572,20.754,153.441
C08612=1083.678,80.881,436.186,174.573,20.756,153.441
C08613=1083.683,81.130,436.168,174.575,20.759,153.442
C08614=1083.689,81.380,436.150,174.577,20.761,153.442
C08615=1083.695,81.629,436.134,174.579,20.762,153.442
C08616=1083.700,81.878,436.116,174.580,20.764,153.442
C08617=1083.706,82.127,436.098,174.582,20.766,153.442
C08618=1083.712,82.377,436.081,174.584,20.769,153.442
C08619=1083.717,82.626,436.063,174.585,20.770,153.442
C08620=1083.723,82.876,436.046,174.587,20.773,153.442
C08621=1083.728,83.125,436.029,174.589,20.775,153.443
C08622=1083.734,83.375,436.011,174.591,20.777,153.443
C08623=1083.740,83.624,435.993,174.592,20.779,153.443
C08624=1083.746,83.872,435.976,174.595,20.781,153.443
C08625=1083.752,84.122,435.958,174.596,20.783,153.443
C08626=1083.758,84.371,435.941,174.598,20.785,153.443
C08627=1083.763,84.621,435.924,174.600,20.787,153.443
C08628=1083.768,84.870,435.906,174.602,20.789,153.443
C08629=1083.774,85.120,435.888,174.603,20.791,153.444
C08630=1083.780,85.369,435.871,174.605,20.793,153.444
C08631=1083.785,85.618,435.853,174.607,20.795,153.444
C08632=1083.792,85.868,435.835,174.609,20.798,153.444
C08633=1083.797,86.117,435.818,174.610,20.800,153.444
C08634=1083.803,86.366,435.800,174.613,20.801,153.444
C08635=1083.809,86.615,435.782,174.614,20.803,153.444
C08636=1083.814,86.864,435.765,174.616,20.806,153.444
C08637=1083.820,87.113,435.747,174.618,20.807,153.444
C08638=1083.826,87.363,435.729,174.620,20.810,153.445
C08639=1083.831,87.612,435.711,174.621,20.812,153.445
C08640=1083.837,87.861,435.694,174.624,20.814,153.445
C08641=1083.843,88.111,435.676,174.625,20.816,153.445
C08642=1083.849,88.360,435.658,174.627,20.818,153.445
C08643=1083.855,88.610,435.640,174.629,20.819,153.445
C08644=1083.860,88.859,435.623,174.631,20.822,153.445
C08645=1083.865,89.108,435.605,174.632,20.823,153.445
C08646=1083.871,89.358,435.587,174.634,20.826,153.445
C08647=1083.877,89.607,435.569,174.636,20.828,153.446
C08648=1083.883,89.857,435.551,174.638,20.830,153.446
C08649=1083.888,90.106,435.534,174.639,20.832,153.446
C08650=1083.894,90.355,435.516,174.642,20.834,153.446
C08651=1083.900,90.604,435.498,174.643,20.835,153.446
C08652=1083.905,90.854,435.481,174.645,20.838,153.446
C08653=1083.912,91.103,435.463,174.647,20.839,153.446
C08654=1083.917,91.352,435.445,174.649,20.842,153.446
C08655=1083.923,91.601,435.428,174.650,20.844,153.446
C08656=1083.928,91.851,435.408,174.653,20.846,153.446
C08657=1083.934,92.100,435.391,174.654,20.848,153.447
C08658=1083.939,92.349,435.373,174.656,20.850,153.447
C08659=1083.945,92.599,435.355,174.658,20.851,153.447
C08660=1083.950,92.848,435.337,174.660,20.854,153.447
C08661=1083.956,93.098,435.319,174.661,20.856,153.447
C08662=1083.962,93.346,435.301,174.663,20.858,153.447
C08663=1083.968,93.595,435.283,174.665,20.860,153.447
C08664=1083.973,93.845,435.265,174.667,20.862,153.448
C08665=1083.979,94.094,435.247,174.668,20.864,153.448
C08666=1083.985,94.344,435.229,174.671,20.866,153.448
C08667=1083.990,94.593,435.210,174.672,20.868,153.448
C08668=1083.996,94.842,435.192,174.674,20.870,153.448
C08669=1084.002,95.121,435.173,174.677,20.872,153.448
C08670=1084.008,95.400,435.152,174.678,20.874,153.448
C08671=1084.015,95.679,435.132,174.680,20.877,153.448
C08672=1084.021,95.959,435.112,174.682,20.879,153.448
C08673=1084.027,96.207,435.094,174.685,20.881,153.448
C08674=1084.033,96.457,435.076,174.686,20.883,153.449
C08675=1084.038,96.706,435.058,174.688,20.885,153.449
C08676=1084.044,96.956,435.039,174.690,20.887,153.449
C08677=1084.050,97.204,435.021,174.692,20.889,153.449
C08678=1084.056,97.454,435.003,174.693,20.891,153.449
C08679=1084.060,97.703,434.985,174.696,20.893,153.449
C08680=1084.067,97.953,434.966,174.697,20.895,153.449
C08681=1084.072,98.202,434.949,174.699,20.896,153.449
C08682=1084.078,98.452,434.930,174.701,20.898,153.449
C08683=1084.084,98.700,434.912,174.703,20.901,153.450
C08684=1084.090,98.950,434.894,174.704,20.902,153.450
C08685=1084.095,99.199,434.875,174.707,20.905,153.450
C08686=1084.101,99.448,434.857,174.708,20.906,153.450
C08687=1084.106,99.697,434.840,174.710,20.909,153.450
C08688=1084.112,99.947,434.821,174.713,20.910,153.450
C08689=1084.118,100.196,434.803,174.714,20.912,153.450
C08690=1084.124,100.445,434.784,174.716,20.914,153.450
C08691=1084.129,100.694,434.766,174.718,20.916,153.450
C08692=1084.135,100.943,434.748,174.720,20.918,153.450
C08693=1084.141,101.192,434.730,174.721,20.920,153.450
C08694=1084.146,101.442,434.711,174.724,20.922,153.450
C08695=1084.152,101.691,434.693,174.725,20.924,153.451
C08696=1084.157,101.941,434.675,174.727,20.926,153.451
C08697=1084.162,102.190,434.656,174.729,20.928,153.451
C08698=1084.169,102.439,434.638,174.731,20.930,153.451
C08699=1084.174,102.689,434.619,174.733,20.932,153.451
C08700=1084.180,102.938,434.601,174.735,20.934,153.451
C08701=1084.185,103.187,434.582,174.737,20.936,153.451
C08702=1084.191,103.436,434.563,174.739,20.937,153.451
C08703=1084.197,103.686,434.545,174.741,20.940,153.451
C08704=1084.202,103.934,434.527,174.742,20.942,153.452
C08705=1084.208,104.184,434.508,174.744,20.944,153.452
C08706=1084.214,104.433,434.490,174.746,20.946,153.452
C08707=1084.219,104.683,434.471,174.748,20.948,153.452
C08708=1084.224,104.931,434.452,174.750,20.950,153.452
C08709=1084.231,105.181,434.434,174.752,20.951,153.452
C08710=1084.236,105.431,434.415,174.754,20.954,153.452
C08711=1084.242,105.679,434.397,174.756,20.955,153.452
C08712=1084.247,105.929,434.378,174.758,20.957,153.452
C08713=1084.253,106.178,434.360,174.759,20.959,153.452
C08714=1084.259,106.427,434.341,174.762,20.961,153.452
C08715=1084.264,106.677,434.322,174.763,20.963,153.452
C08716=1084.270,106.925,434.304,174.765,20.965,153.452
C08717=1084.276,107.175,434.285,174.768,20.967,153.453
C08718=1084.281,107.424,434.267,174.769,20.969,153.453
C08719=1084.287,107.673,434.248,174.771,20.971,153.453
C08720=1084.292,107.923,434.229,174.773,20.973,153.453
C08721=1084.298,108.172,434.211,174.775,20.975,153.453
C08722=1084.304,108.421,434.192,174.776,20.977,153.453
C08723=1084.310,108.670,434.173,174.779,20.978,153.453
C08724=1084.315,108.919,434.154,174.781,20.981,153.453
C08725=1084.321,109.169,434.136,174.783,20.982,153.453
C08726=1084.327,109.418,434.117,174.785,20.985,153.453
C08727=1084.332,109.667,434.098,174.786,20.986,153.453
C08728=1084.338,109.916,434.079,174.789,20.988,153.453
C08729=1084.344,110.166,434.061,174.791,20.990,153.454
C08730=1084.349,110.415,434.042,174.792,20.992,153.454
C08731=1084.355,110.664,434.023,174.795,20.994,153.454
C08732=1084.361,110.913,434.004,174.796,20.996,153.454
C08733=1084.367,111.192,433.983,174.799,20.998,153.454
C08734=1084.374,111.471,433.962,174.801,21.000,153.454
C08735=1084.380,111.750,433.941,174.803,21.002,153.454
C08736=1084.386,112.029,433.920,174.805,21.004,153.454
C08737=1084.391,112.279,433.902,174.807,21.006,153.454
C08738=1084.398,112.528,433.883,174.809,21.008,153.454
C08739=1084.403,112.777,433.864,174.811,21.010,153.454
C08740=1084.409,113.027,433.845,174.813,21.012,153.454
C08741=1084.414,113.276,433.826,174.815,21.014,153.454
C08742=1084.419,113.525,433.807,174.817,21.015,153.455
C08743=1084.426,113.774,433.788,174.819,21.018,153.455
C08744=1084.432,114.023,433.769,174.821,21.020,153.455
C08745=1084.437,114.273,433.750,174.823,21.021,153.455
C08746=1084.442,114.521,433.731,174.825,21.024,153.455
C08747=1084.448,114.771,433.712,174.826,21.025,153.455
C08748=1084.453,115.021,433.693,174.829,21.027,153.455
C08749=1084.458,115.270,433.674,174.831,21.029,153.455
C08750=1084.464,115.519,433.655,174.833,21.031,153.455
C08751=1084.470,115.768,433.636,174.835,21.033,153.455
C08752=1084.476,116.017,433.617,174.836,21.035,153.455
C08753=1084.481,116.266,433.598,174.838,21.037,153.455
C08754=1084.487,116.516,433.579,174.841,21.039,153.455
C08755=1084.492,116.764,433.560,174.842,21.040,153.455
C08756=1084.498,117.014,433.541,174.845,21.043,153.456
C08757=1084.504,117.263,433.521,174.846,21.044,153.456
C08758=1084.509,117.513,433.502,174.848,21.047,153.456
C08759=1084.515,117.761,433.483,174.851,21.049,153.456
C08760=1084.520,118.010,433.463,174.852,21.050,153.456
C08761=1084.526,118.260,433.444,174.854,21.052,153.456
C08762=1084.532,118.509,433.425,174.857,21.054,153.456
C08763=1084.537,118.758,433.406,174.858,21.056,153.456
C08764=1084.542,119.007,433.387,174.860,21.058,153.456
C08765=1084.548,119.257,433.367,174.862,21.060,153.456
C08766=1084.554,119.506,433.348,174.864,21.062,153.456
C08767=1084.559,119.755,433.329,174.867,21.064,153.456
C08768=1084.565,120.004,433.310,174.868,21.065,153.456
C08769=1084.571,120.253,433.290,174.871,21.067,153.456
C08770=1084.576,120.503,433.271,174.873,21.070,153.457
C08771=1084.581,120.751,433.252,174.874,21.071,153.457
C08772=1084.586,121.001,433.232,174.877,21.073,153.457
C08773=1084.592,121.251,433.213,174.878,21.075,153.457
C08774=1084.598,121.500,433.194,174.880,21.077,153.457
C08775=1084.604,121.749,433.174,174.883,21.079,153.457
C08776=1084.609,121.998,433.155,174.884,21.080,153.457
C08777=1084.614,122.247,433.136,174.886,21.083,153.457
C08778=1084.620,122.496,433.116,174.889,21.084,153.457
C08779=1084.626,122.745,433.096,174.890,21.086,153.457
C08780=1084.632,122.995,433.077,174.893,21.088,153.457
C08781=1084.637,123.244,433.058,174.895,21.090,153.457
C08782=1084.643,123.493,433.039,174.897,21.092,153.457
C08783=1084.649,123.742,433.019,174.899,21.094,153.457
C08784=1084.654,123.991,433.000,174.900,21.095,153.457
C08785=1084.660,124.240,432.981,174.903,21.097,153.457
C08786=1084.666,124.489,432.961,174.905,21.099,153.458
C08787=1084.672,124.739,432.941,174.907,21.101,153.458
C08788=1084.677,124.988,432.922,174.909,21.103,153.458
C08789=1084.683,125.237,432.902,174.911,21.105,153.458
C08790=1084.688,125.486,432.883,174.913,21.106,153.458
C08791=1084.693,125.735,432.863,174.915,21.108,153.458
C08792=1084.699,125.984,432.844,174.917,21.110,153.458
C08793=1084.705,126.234,432.824,174.919,21.112,153.458
C08794=1084.711,126.483,432.805,174.921,21.114,153.458
C08795=1084.717,126.732,432.785,174.924,21.116,153.458
C08796=1084.722,126.981,432.766,174.925,21.117,153.458
C08797=1084.728,127.260,432.743,174.928,21.119,153.458
C08798=1084.735,127.540,432.722,174.930,21.121,153.458
C08799=1084.741,127.818,432.700,174.932,21.123,153.458
C08800=1084.748,128.098,432.678,174.935,21.126,153.458
C08801=1084.754,128.347,432.658,174.937,21.127,153.458
C08802=1084.759,128.596,432.638,174.939,21.129,153.458
C08803=1084.765,128.845,432.618,174.941,21.131,153.458
C08804=1084.770,129.095,432.599,174.943,21.133,153.458
C08805=1084.776,129.343,432.579,174.946,21.135,153.458
C08806=1084.781,129.592,432.560,174.947,21.136,153.458
C08807=1084.787,129.841,432.540,174.950,21.138,153.458
C08808=1084.792,130.091,432.520,174.952,21.140,153.458
C08809=1084.798,130.340,432.500,174.953,21.142,153.459
C08810=1084.804,130.589,432.481,174.956,21.144,153.459
C08811=1084.810,130.838,432.461,174.958,21.146,153.459
C08812=1084.816,131.087,432.441,174.960,21.147,153.459
C08813=1084.822,131.336,432.422,174.962,21.149,153.459
C08814=1084.828,131.586,432.401,174.964,21.151,153.459
C08815=1084.833,131.835,432.382,174.966,21.152,153.459
C08816=1084.839,132.084,432.362,174.968,21.154,153.459
C08817=1084.845,132.334,432.343,174.971,21.156,153.459
C08818=1084.850,132.583,432.322,174.972,21.157,153.459
C08819=1084.856,132.831,432.303,174.975,21.159,153.459
C08820=1084.861,133.080,432.283,174.977,21.161,153.459
C08821=1084.867,133.329,432.263,174.978,21.163,153.459
C08822=1084.873,133.578,432.243,174.981,21.165,153.459
C08823=1084.877,133.828,432.223,174.983,21.167,153.459
C08824=1084.883,134.077,432.203,174.986,21.169,153.459
C08825=1084.889,134.326,432.183,174.987,21.170,153.459
C08826=1084.894,134.575,432.163,174.990,21.172,153.459
C08827=1084.900,134.824,432.143,174.992,21.174,153.459
C08828=1084.906,135.073,432.123,174.994,21.175,153.459
C08829=1084.911,135.323,432.103,174.996,21.177,153.459
C08830=1084.917,135.572,432.083,174.998,21.180,153.459
C08831=1084.923,135.821,432.063,175.000,21.181,153.459
C08832=1084.929,136.070,432.043,175.002,21.183,153.459
C08833=1084.934,136.320,432.023,175.004,21.185,153.459
C08834=1084.940,136.569,432.003,175.007,21.187,153.459
C08835=1084.945,136.818,431.982,175.008,21.188,153.459
C08836=1084.951,137.067,431.962,175.011,21.190,153.459
C08837=1084.956,137.316,431.942,175.013,21.192,153.459
C08838=1084.962,137.565,431.923,175.015,21.194,153.459
C08839=1084.968,137.814,431.902,175.017,21.195,153.459
C08840=1084.974,138.063,431.882,175.020,21.197,153.459
C08841=1084.979,138.312,431.861,175.022,21.199,153.459
C08842=1084.985,138.561,431.841,175.023,21.201,153.459
C08843=1084.990,138.811,431.822,175.026,21.203,153.459
C08844=1084.996,139.060,431.802,175.028,21.204,153.459
C08845=1085.001,139.309,431.781,175.030,21.206,153.460
C08846=1085.008,139.558,431.761,175.032,21.208,153.460
C08847=1085.013,139.807,431.740,175.035,21.210,153.460
C08848=1085.019,140.056,431.720,175.037,21.212,153.460
C08849=1085.024,140.305,431.700,175.039,21.213,153.460
C08850=1085.030,140.554,431.680,175.041,21.215,153.460
C08851=1085.035,140.803,431.659,175.043,21.217,153.460
C08852=1085.041,141.052,431.639,175.045,21.218,153.460
C08853=1085.046,141.302,431.619,175.047,21.220,153.460
C08854=1085.052,141.551,431.599,175.050,21.222,153.460
C08855=1085.057,141.800,431.578,175.052,21.224,153.460
C08856=1085.063,142.050,431.558,175.054,21.225,153.460
C08857=1085.069,142.299,431.537,175.056,21.227,153.460
C08858=1085.075,142.547,431.517,175.058,21.229,153.460
C08859=1085.080,142.797,431.497,175.061,21.231,153.460
C08860=1085.085,143.046,431.476,175.062,21.232,153.460
C08861=1085.092,143.324,431.453,175.065,21.234,153.460
C08862=1085.098,143.603,431.430,175.068,21.237,153.460
C08863=1085.104,143.882,431.408,175.070,21.239,153.460
C08864=1085.111,144.161,431.384,175.073,21.241,153.460
C08865=1085.116,144.410,431.364,175.074,21.242,153.460
C08866=1085.122,144.659,431.344,175.077,21.244,153.460
C08867=1085.127,144.908,431.323,175.079,21.246,153.460
C08868=1085.133,145.157,431.303,175.082,21.247,153.460
C08869=1085.138,145.407,431.282,175.083,21.249,153.460
C08870=1085.144,145.656,431.262,175.086,21.251,153.460
C08871=1085.150,145.905,431.241,175.088,21.253,153.460
C08872=1085.155,146.154,431.221,175.090,21.255,153.460
C08873=1085.161,146.403,431.201,175.092,21.256,153.460
C08874=1085.167,146.652,431.179,175.094,21.258,153.460
C08875=1085.172,146.901,431.158,175.097,21.260,153.460
C08876=1085.178,147.150,431.138,175.099,21.262,153.460
C08877=1085.184,147.399,431.118,175.102,21.264,153.460
C08878=1085.189,147.648,431.097,175.103,21.265,153.460
C08879=1085.195,147.898,431.076,175.106,21.266,153.460
C08880=1085.200,148.147,431.055,175.108,21.268,153.460
C08881=1085.206,148.395,431.035,175.111,21.270,153.460
C08882=1085.212,148.645,431.015,175.112,21.272,153.460
C08883=1085.218,148.894,430.993,175.114,21.273,153.460
C08884=1085.223,149.143,430.972,175.117,21.275,153.460
C08885=1085.228,149.392,430.952,175.119,21.277,153.460
C08886=1085.234,149.641,430.931,175.121,21.279,153.460
C08887=1085.240,149.889,430.911,175.123,21.281,153.460
C08888=1085.246,150.139,430.890,175.126,21.282,153.460
C08889=1085.251,150.388,430.869,175.128,21.284,153.460
C08890=1085.256,150.637,430.849,175.131,21.286,153.460
C08891=1085.262,150.886,430.827,175.132,21.287,153.460
C08892=1085.268,151.136,430.806,175.135,21.289,153.460
C08893=1085.273,151.385,430.786,175.137,21.291,153.460
C08894=1085.278,151.633,430.765,175.139,21.293,153.460
C08895=1085.284,151.882,430.744,175.142,21.295,153.460
C08896=1085.290,152.132,430.722,175.143,21.296,153.460
C08897=1085.295,152.381,430.702,175.146,21.298,153.460
C08898=1085.300,152.630,430.681,175.148,21.300,153.460
C08899=1085.307,152.879,430.660,175.151,21.301,153.460
C08900=1085.313,153.128,430.640,175.153,21.303,153.460
C08901=1085.318,153.376,430.619,175.155,21.305,153.460
C08902=1085.323,153.626,430.598,175.157,21.306,153.460
C08903=1085.329,153.875,430.577,175.160,21.308,153.460
C08904=1085.335,154.124,430.556,175.162,21.310,153.460
C08905=1085.340,154.373,430.535,175.165,21.312,153.460
C08906=1085.346,154.622,430.514,175.166,21.313,153.460
C08907=1085.351,154.871,430.493,175.169,21.315,153.460
C08908=1085.357,155.120,430.472,175.171,21.317,153.460
C08909=1085.363,155.370,430.451,175.173,21.319,153.460
C08910=1085.368,155.618,430.430,175.176,21.320,153.460
C08911=1085.374,155.867,430.409,175.178,21.322,153.460
C08912=1085.380,156.117,430.387,175.180,21.323,153.460
C08913=1085.385,156.366,430.367,175.182,21.325,153.460
C08914=1085.390,156.614,430.345,175.185,21.327,153.460
C08915=1085.396,156.864,430.323,175.187,21.329,153.460
C08916=1085.401,157.113,430.303,175.190,21.330,153.460
C08917=1085.407,157.361,430.282,175.191,21.332,153.460
C08918=1085.413,157.611,430.261,175.194,21.334,153.460
C08919=1085.418,157.860,430.239,175.196,21.336,153.460
C08920=1085.424,158.109,430.218,175.199,21.338,153.460
C08921=1085.430,158.358,430.197,175.201,21.339,153.460
C08922=1085.435,158.606,430.176,175.204,21.341,153.460
C08923=1085.441,158.856,430.155,175.205,21.342,153.460
C08924=1085.446,159.105,430.133,175.208,21.344,153.460
C08925=1085.453,159.384,430.110,175.210,21.346,153.460
C08926=1085.459,159.663,430.085,175.213,21.348,153.460
C08927=1085.465,159.942,430.062,175.216,21.350,153.460
C08928=1085.471,160.220,430.038,175.218,21.352,153.460
C08929=1085.477,160.469,430.017,175.221,21.354,153.460
C08930=1085.482,160.718,429.995,175.223,21.355,153.460
C08931=1085.489,160.967,429.974,175.225,21.356,153.460
C08932=1085.494,161.216,429.953,175.227,21.358,153.460
C08933=1085.500,161.465,429.932,175.230,21.360,153.460
C08934=1085.505,161.714,429.910,175.232,21.362,153.460
C08935=1085.510,161.962,429.888,175.234,21.364,153.460
C08936=1085.516,162.213,429.867,175.237,21.365,153.460
C08937=1085.521,162.461,429.846,175.239,21.367,153.460
C08938=1085.527,162.709,429.824,175.241,21.369,153.460
C08939=1085.532,162.959,429.802,175.243,21.370,153.460
C08940=1085.538,163.208,429.781,175.246,21.372,153.460
C08941=1085.543,163.458,429.759,175.248,21.374,153.460
C08942=1085.548,163.706,429.738,175.251,21.376,153.460
C08943=1085.554,163.955,429.717,175.253,21.377,153.460
C08944=1085.559,164.204,429.695,175.256,21.379,153.460
C08945=1085.565,164.453,429.673,175.257,21.381,153.460
C08946=1085.570,164.702,429.651,175.260,21.383,153.460
C08947=1085.576,164.951,429.630,175.262,21.385,153.460
C08948=1085.581,165.200,429.608,175.264,21.386,153.460
C08949=1085.587,165.449,429.587,175.267,21.388,153.460
C08950=1085.591,165.698,429.565,175.269,21.390,153.460
C08951=1085.598,165.947,429.544,175.272,21.392,153.460
C08952=1085.602,166.196,429.522,175.274,21.393,153.460
C08953=1085.609,166.445,429.500,175.277,21.395,153.460
C08954=1085.613,166.694,429.478,175.278,21.396,153.460
C08955=1085.620,166.943,429.457,175.281,21.398,153.460
C08956=1085.625,167.192,429.435,175.283,21.400,153.460
C08957=1085.630,167.441,429.413,175.286,21.402,153.460
C08958=1085.636,167.690,429.392,175.288,21.403,153.460
C08959=1085.641,167.939,429.370,175.291,21.405,153.460
C08960=1085.647,168.188,429.348,175.293,21.407,153.460
C08961=1085.652,168.437,429.326,175.296,21.409,153.460
C08962=1085.658,168.686,429.305,175.298,21.410,153.460
C08963=1085.663,168.935,429.283,175.300,21.412,153.460
C08964=1085.669,169.184,429.261,175.302,21.414,153.460
C08965=1085.674,169.433,429.239,175.305,21.415,153.460
C08966=1085.679,169.682,429.217,175.307,21.417,153.460
C08967=1085.686,169.931,429.195,175.310,21.419,153.460
C08968=1085.691,170.180,429.173,175.312,21.421,153.460
C08969=1085.697,170.429,429.151,175.315,21.422,153.460
C08970=1085.702,170.678,429.129,175.317,21.424,153.460
C08971=1085.708,170.927,429.108,175.319,21.426,153.460
C08972=1085.713,171.176,429.086,175.322,21.428,153.460
C08973=1085.719,171.425,429.064,175.324,21.429,153.460
C08974=1085.724,171.673,429.042,175.326,21.430,153.460
C08975=1085.730,171.922,429.020,175.328,21.432,153.460
C08976=1085.735,172.172,428.998,175.331,21.434,153.459
C08977=1085.740,172.421,428.976,175.333,21.436,153.459
C08978=1085.746,172.670,428.954,175.336,21.437,153.460
C08979=1085.752,172.918,428.932,175.338,21.439,153.459
C08980=1085.758,173.167,428.910,175.341,21.441,153.459
C08981=1085.763,173.417,428.888,175.344,21.442,153.459
C08982=1085.769,173.665,428.867,175.346,21.444,153.459
C08983=1085.774,173.914,428.844,175.348,21.446,153.459
C08984=1085.779,174.163,428.822,175.351,21.447,153.459
C08985=1085.785,174.412,428.800,175.353,21.449,153.459
C08986=1085.791,174.662,428.778,175.356,21.451,153.459
C08987=1085.797,174.910,428.756,175.358,21.452,153.459
C08988=1085.802,175.159,428.734,175.360,21.454,153.459
C08989=1085.808,175.438,428.709,175.363,21.456,153.459
C08990=1085.815,175.716,428.684,175.366,21.458,153.459
C08991=1085.821,175.994,428.659,175.368,21.459,153.459
C08992=1085.827,176.273,428.635,175.372,21.461,153.459
C08993=1085.832,176.522,428.613,175.374,21.463,153.459
C08994=1085.839,176.770,428.590,175.376,21.465,153.459
C08995=1085.844,177.020,428.568,175.378,21.466,153.459
C08996=1085.850,177.268,428.546,175.381,21.468,153.459
C08997=1085.855,177.517,428.524,175.383,21.469,153.459
C08998=1085.861,177.767,428.502,175.386,21.471,153.459
C08999=1085.867,178.015,428.479,175.388,21.472,153.459
C09000=1085.872,178.264,428.457,175.391,21.474,153.459
C09001=1085.878,178.513,428.435,175.393,21.476,153.459
C09002=1085.884,178.762,428.413,175.396,21.478,153.459
C09003=1085.890,179.011,428.390,175.398,21.479,153.458
C09004=1085.894,179.260,428.368,175.401,21.481,153.458
C09005=1085.901,179.508,428.346,175.404,21.482,153.458
C09006=1085.906,179.758,428.323,175.406,21.484,153.458
C09007=1085.912,180.007,428.301,175.409,21.485,153.458
C09008=1085.918,180.256,428.278,175.411,21.487,153.458
C09009=1085.923,180.504,428.256,175.414,21.489,153.458
C09010=1085.929,180.754,428.234,175.416,21.491,153.458
C09011=1085.935,181.003,428.211,175.419,21.492,153.458
C09012=1085.941,181.251,428.189,175.421,21.494,153.458
C09013=1085.946,181.501,428.167,175.424,21.495,153.458
C09014=1085.952,181.749,428.144,175.426,21.497,153.458
C09015=1085.957,181.998,428.122,175.429,21.498,153.458
C09016=1085.963,182.247,428.099,175.431,21.500,153.458
C09017=1085.969,182.496,428.076,175.434,21.502,153.458
C09018=1085.975,182.745,428.054,175.436,21.504,153.458
C09019=1085.980,182.993,428.032,175.439,21.505,153.458
C09020=1085.986,183.242,428.009,175.441,21.507,153.458
C09021=1085.992,183.492,427.987,175.444,21.508,153.458
C09022=1085.997,183.741,427.964,175.446,21.510,153.457
C09023=1086.004,183.989,427.942,175.449,21.511,153.457
C09024=1086.009,184.239,427.920,175.451,21.513,153.457
C09025=1086.015,184.488,427.897,175.454,21.515,153.457
C09026=1086.021,184.736,427.874,175.456,21.516,153.457
C09027=1086.026,184.985,427.851,175.459,21.517,153.457
C09028=1086.031,185.234,427.829,175.462,21.519,153.457
C09029=1086.037,185.483,427.806,175.464,21.521,153.457
C09030=1086.043,185.732,427.783,175.467,21.523,153.457
C09031=1086.048,185.981,427.760,175.469,21.525,153.457
C09032=1086.053,186.230,427.738,175.471,21.526,153.457
C09033=1086.059,186.479,427.715,175.474,21.528,153.457
C09034=1086.065,186.727,427.692,175.476,21.530,153.457
C09035=1086.070,186.976,427.669,175.479,21.531,153.457
C09036=1086.076,187.225,427.647,175.481,21.533,153.457
C09037=1086.081,187.474,427.623,175.484,21.535,153.457
C09038=1086.086,187.723,427.601,175.487,21.536,153.457
C09039=1086.092,187.972,427.578,175.489,21.538,153.457
C09040=1086.098,188.221,427.555,175.492,21.539,153.457
C09041=1086.103,188.469,427.532,175.494,21.541,153.457
C09042=1086.108,188.718,427.510,175.496,21.543,153.457
C09043=1086.113,188.967,427.486,175.499,21.545,153.457
C09044=1086.119,189.216,427.463,175.501,21.546,153.457
C09045=1086.125,189.465,427.440,175.504,21.548,153.457
C09046=1086.131,189.714,427.417,175.506,21.550,153.457
C09047=1086.136,189.963,427.394,175.509,21.551,153.456
C09048=1086.141,190.211,427.372,175.512,21.553,153.456
C09049=1086.146,190.461,427.349,175.514,21.555,153.456
C09050=1086.152,190.710,427.326,175.517,21.556,153.456
C09051=1086.158,190.959,427.303,175.520,21.558,153.456
C09052=1086.163,191.208,427.280,175.522,21.560,153.456
C09053=1086.169,191.486,427.254,175.525,21.562,153.456
C09054=1086.176,191.763,427.228,175.528,21.563,153.456
C09055=1086.182,192.042,427.202,175.531,21.565,153.456
C09056=1086.188,192.319,427.177,175.533,21.567,153.456
C09057=1086.194,192.568,427.154,175.536,21.569,153.456
C09058=1086.199,192.817,427.130,175.538,21.571,153.456
C09059=1086.205,193.066,427.107,175.541,21.572,153.456
C09060=1086.210,193.315,427.084,175.544,21.574,153.456
C09061=1086.216,193.563,427.061,175.547,21.576,153.456
C09062=1086.221,193.813,427.037,175.549,21.578,153.456
C09063=1086.227,194.062,427.014,175.552,21.579,153.456
C09064=1086.233,194.310,426.991,175.554,21.581,153.456
C09065=1086.238,194.559,426.969,175.557,21.582,153.456
C09066=1086.243,194.808,426.945,175.559,21.584,153.456
C09067=1086.249,195.057,426.922,175.562,21.585,153.455
C09068=1086.255,195.305,426.899,175.565,21.587,153.455
C09069=1086.260,195.554,426.876,175.567,21.589,153.455
C09070=1086.265,195.803,426.852,175.570,21.590,153.455
C09071=1086.271,196.052,426.829,175.572,21.592,153.455
C09072=1086.277,196.300,426.805,175.575,21.594,153.455
C09073=1086.282,196.550,426.782,175.578,21.596,153.455
C09074=1086.289,196.799,426.759,175.581,21.597,153.455
C09075=1086.294,197.048,426.736,175.583,21.599,153.455
C09076=1086.300,197.296,426.712,175.586,21.600,153.455
C09077=1086.305,197.546,426.688,175.588,21.602,153.455
C09078=1086.311,197.794,426.665,175.591,21.604,153.455
C09079=1086.317,198.043,426.642,175.593,21.605,153.455
C09080=1086.322,198.292,426.618,175.596,21.607,153.455
C09081=1086.328,198.541,426.595,175.598,21.608,153.455
C09082=1086.334,198.789,426.572,175.602,21.610,153.455
C09083=1086.339,199.038,426.548,175.604,21.612,153.455
C09084=1086.345,199.287,426.525,175.607,21.613,153.454
C09085=1086.351,199.535,426.502,175.609,21.615,153.454
C09086=1086.356,199.785,426.478,175.612,21.616,153.454
C09087=1086.361,200.034,426.455,175.614,21.618,153.454
C09088=1086.368,200.283,426.431,175.617,21.620,153.454
C09089=1086.373,200.532,426.407,175.620,21.621,153.454
C09090=1086.379,200.780,426.384,175.623,21.623,153.454
C09091=1086.385,201.029,426.361,175.625,21.625,153.454
C09092=1086.390,201.278,426.337,175.628,21.627,153.454
C09093=1086.396,201.526,426.314,175.630,21.628,153.454
C09094=1086.401,201.775,426.289,175.633,21.629,153.454
C09095=1086.407,202.025,426.266,175.636,21.631,153.454
C09096=1086.413,202.273,426.242,175.638,21.633,153.454
C09097=1086.418,202.522,426.219,175.641,21.634,153.454
C09098=1086.424,202.770,426.195,175.644,21.636,153.454
C09099=1086.429,203.020,426.172,175.647,21.638,153.453
C09100=1086.436,203.268,426.148,175.649,21.640,153.454
C09101=1086.441,203.517,426.124,175.652,21.641,153.453
C09102=1086.446,203.766,426.100,175.654,21.643,153.453
C09103=1086.452,204.015,426.077,175.657,21.644,153.453
C09104=1086.457,204.264,426.053,175.659,21.646,153.453
C09105=1086.463,204.512,426.029,175.663,21.648,153.453
C09106=1086.468,204.761,426.005,175.665,21.650,153.453
